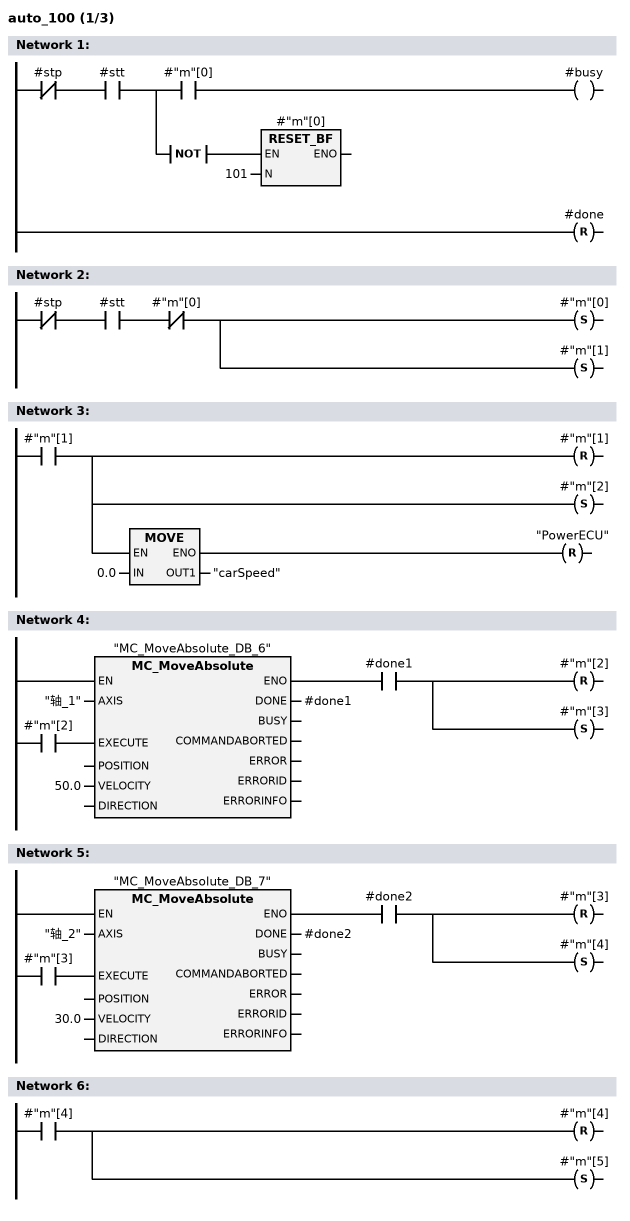
   // no SCL statement known for RBitfield: written as a call
   #_w1 := NOT #stp AND #stt;
   #busy := #_w1 AND #"m"[0];
   IF NOT #_w1 THEN RESET_BF(operand := #"m"[0], n := 101); END_IF;
   #done := FALSE;
END_REGION

REGION Network 2
   RUNG wire#powerrail
      I_Contact( #stp )
      Contact( #stt )
      I_Contact( #"m"[0] )
      wire#w1
      S_Coil( #"m"[0] )
   END_RUNG
   RUNG wire#w1
      S_Coil( #"m"[1] )
   END_RUNG
   // the same network as SCL:
   #_w1 := NOT #stp AND #stt AND NOT #"m"[0];
   IF #_w1 THEN
       #"m"[0] := TRUE;
       #"m"[1] := TRUE;
   END_IF;
END_REGION

REGION Network 3
   RUNG wire#powerrail
      Contact( #"m"[1] )
      wire#w1
      R_Coil( #"m"[1] )
   END_RUNG
   RUNG wire#w1
      S_Coil( #"m"[2] )
   END_RUNG
   RUNG wire#w1
      Move(in := 0.0, out1 => "carSpeed")
      R_Coil( "PowerECU" )
   END_RUNG
   // the same network as SCL:
   #_w1 := #"m"[1];
   IF #_w1 THEN
       #"m"[1] := FALSE;
       #"m"[2] := TRUE;
       "carSpeed" := 0.0;
       "PowerECU" := FALSE;
   END_IF;
END_REGION

REGION Network 4
   // ENO of a box is taken as its EN; it also drops when the box reports an error
   "MC_MoveAbsolute_DB_6"(Axis := "轴_1", Execute := #"m"[2], Velocity := 50.0, Done => #done1);   // MC_MoveAbsolute
   IF #done1 THEN
       #"m"[2] := FALSE;
       #"m"[3] := TRUE;
   END_IF;
END_REGION

REGION Network 5
   // ENO of a box is taken as its EN; it also drops when the box reports an error
   "MC_MoveAbsolute_DB_7"(Axis := "轴_2", Execute := #"m"[3], Velocity := 30.0, Done => #done2);   // MC_MoveAbsolute
   IF #done2 THEN
       #"m"[3] := FALSE;
       #"m"[4] := TRUE;
   END_IF;
END_REGION

REGION Network 6
   RUNG wire#powerrail
      Contact( #"m"[4] )
      wire#w1
      R_Coil( #"m"[4] )
   END_RUNG
   RUNG wire#w1
      S_Coil( #"m"[5] )
   END_RUNG
   // the same network as SCL:
   #_w1 := #"m"[4];
   IF #_w1 THEN
       #"m"[4] := FALSE;
       #"m"[5] := TRUE;
   END_IF;
END_REGION

REGION Network 7
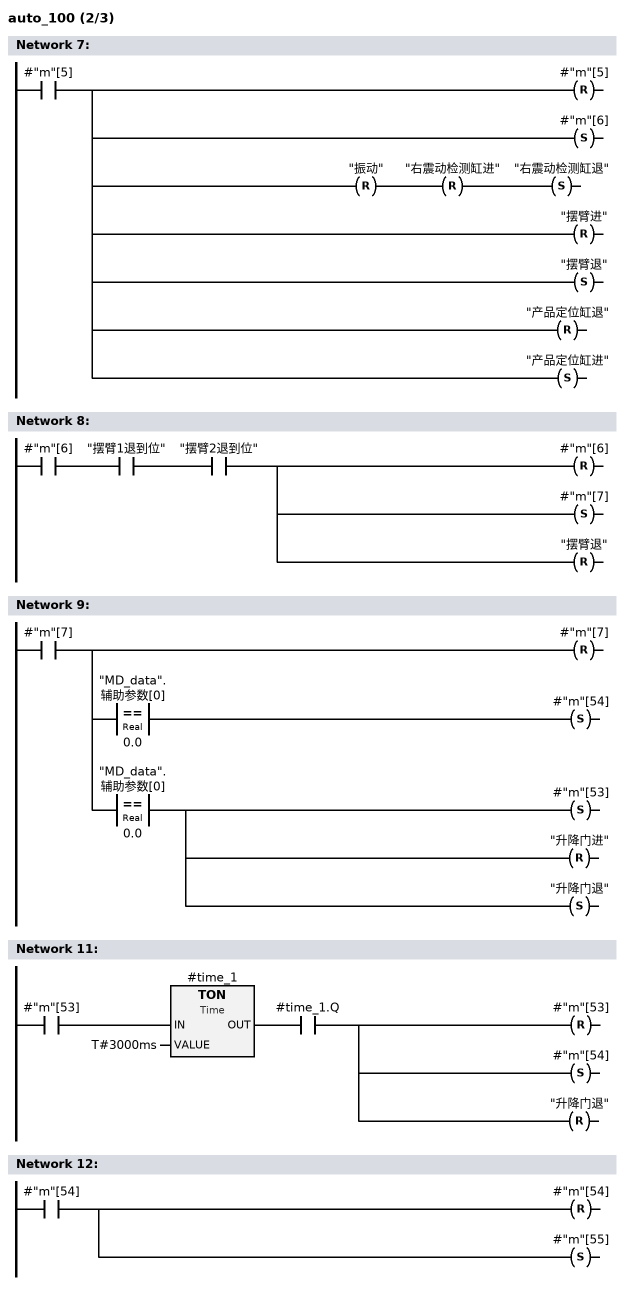
   RUNG wire#powerrail
      Contact( #"m"[5] )
      wire#w1
      R_Coil( #"m"[5] )
   END_RUNG
   RUNG wire#w1
      S_Coil( #"m"[6] )
   END_RUNG
   RUNG wire#w1
      R_Coil( "振动" )
      R_Coil( "右震动检测缸进" )
      S_Coil( "右震动检测缸退" )
   END_RUNG
   RUNG wire#w1
      R_Coil( "摆臂进" )
   END_RUNG
   RUNG wire#w1
      S_Coil( "摆臂退" )
   END_RUNG
   RUNG wire#w1
      R_Coil( "产品定位缸退" )
   END_RUNG
   RUNG wire#w1
      S_Coil( "产品定位缸进" )
   END_RUNG
   // the same network as SCL:
   #_w1 := #"m"[5];
   IF #_w1 THEN
       #"m"[5] := FALSE;
       #"m"[6] := TRUE;
       "振动" := FALSE;
       "右震动检测缸进" := FALSE;
       "右震动检测缸退" := TRUE;
       "摆臂进" := FALSE;
       "摆臂退" := TRUE;
       "产品定位缸退" := FALSE;
       "产品定位缸进" := TRUE;
   END_IF;
END_REGION

REGION Network 8
   RUNG wire#powerrail
      Contact( #"m"[6] )
      Contact( "摆臂1退到位" )
      Contact( "摆臂2退到位" )
      wire#w1
      R_Coil( #"m"[6] )
   END_RUNG
   RUNG wire#w1
      S_Coil( #"m"[7] )
   END_RUNG
   RUNG wire#w1
      R_Coil( "摆臂退" )
   END_RUNG
   // the same network as SCL:
   #_w1 := #"m"[6] AND "摆臂1退到位" AND "摆臂2退到位";
   IF #_w1 THEN
       #"m"[6] := FALSE;
       #"m"[7] := TRUE;
       "摆臂退" := FALSE;
   END_IF;
END_REGION

REGION Network 9
   RUNG wire#powerrail
      Contact( #"m"[7] )
      wire#w1
      R_Coil( #"m"[7] )
   END_RUNG
   RUNG wire#w1
      { S7_Templates := "SrcType := Real" } EQ_Contact(in1 := "MD_data".辅助参数[0], in2 := 0.0)
      S_Coil( #"m"[54] )
   END_RUNG
   RUNG wire#w1
      { S7_Templates := "SrcType := Real" } EQ_Contact(in1 := "MD_data".辅助参数[0], in2 := 0.0)
      wire#w2
      S_Coil( #"m"[53] )
   END_RUNG
   RUNG wire#w2
      R_Coil( "升降门进" )
   END_RUNG
   RUNG wire#w2
      S_Coil( "升降门退" )
   END_RUNG
   // the same network as SCL:
   #_w1 := #"m"[7];
   IF #_w1 THEN #"m"[7] := FALSE; END_IF;
   IF #_w1 AND ("MD_data".辅助参数[0] = 0.0) THEN
       #"m"[54] := TRUE;
       #"m"[53] := TRUE;
       "升降门进" := FALSE;
       "升降门退" := TRUE;
   END_IF;
END_REGION

REGION Network 11
   #time_1.TON(IN := #"m"[53], PT := T#3000ms);   // TON coil
   #_w1 := #"m"[53] AND #time_1.Q;
   IF #_w1 THEN
       #"m"[53] := FALSE;
       #"m"[54] := TRUE;
       "升降门退" := FALSE;
   END_IF;
END_REGION

REGION Network 12
   RUNG wire#powerrail
      Contact( #"m"[54] )
      wire#w1
      R_Coil( #"m"[54] )
   END_RUNG
   RUNG wire#w1
      S_Coil( #"m"[55] )
   END_RUNG
   // the same network as SCL:
   #_w1 := #"m"[54];
   IF #_w1 THEN
       #"m"[54] := FALSE;
       #"m"[55] := TRUE;
   END_IF;
END_REGION

REGION Network 14
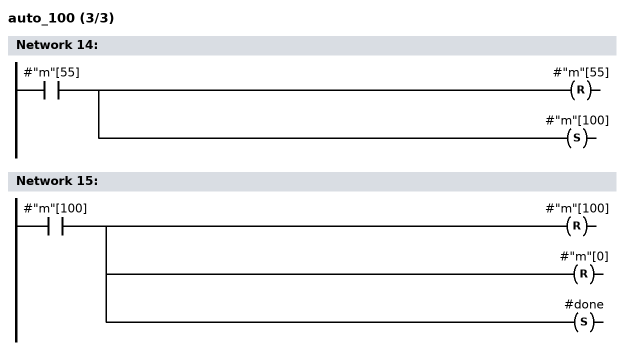
   RUNG wire#powerrail
      Contact( #"m"[55] )
      wire#w1
      R_Coil( #"m"[55] )
   END_RUNG
   RUNG wire#w1
      S_Coil( #"m"[100] )
   END_RUNG
   // the same network as SCL:
   #_w1 := #"m"[55];
   IF #_w1 THEN
       #"m"[55] := FALSE;
       #"m"[100] := TRUE;
   END_IF;
END_REGION

REGION Network 15
   RUNG wire#powerrail
      Contact( #"m"[100] )
      wire#w1
      R_Coil( #"m"[100] )
   END_RUNG
   RUNG wire#w1
      R_Coil( #"m"[0] )
   END_RUNG
   RUNG wire#w1
      S_Coil( #done )
   END_RUNG
   // the same network as SCL:
   #_w1 := #"m"[100];
   IF #_w1 THEN
       #"m"[100] := FALSE;
       #"m"[0] := FALSE;
       #done := TRUE;
   END_IF;
END_REGION
END_FUNCTION_BLOCK

FUNCTION_BLOCK "功能"   // FB14, LAD
{ S7_Optimized_Access := 'TRUE' }
VERSION : 0.1
   VAR_INPUT
      stt : Bool;
      stp : Bool;
      direction : Bool;
      speed : Real;
      angle : Real;
   END_VAR
   VAR_OUTPUT
      done : Bool;
      error : Bool;
      busy : Bool;
   END_VAR
   VAR
      "m" : Array[0..100] of Bool;
      "time" : IEC_TIMER;
      newCV : DInt;
      angleSet : Real;
      speedSet : Real;
      angleRead : Real;
      torqueOutputB : Real;
      loadOutput : Real;
      speedReal : Real;
   END_VAR
   VAR_TEMP   // added for the SCL form of the ladder/FBD networks
      _w1 : Bool;
      _w2 : Bool;
      _w3 : Bool;
      _w4 : Bool;
      _w5 : Bool;
   END_VAR
BEGIN

REGION Network 1
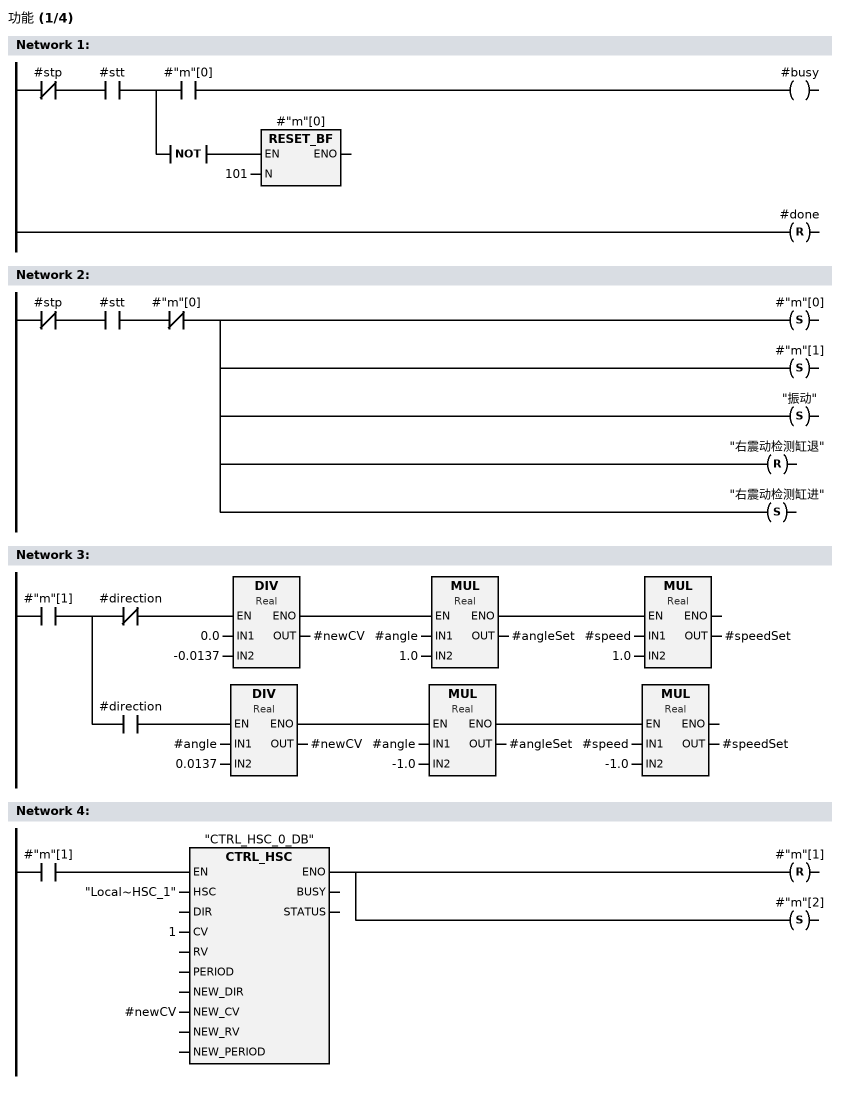
   // no SCL statement known for RBitfield: written as a call
   #_w1 := NOT #stp AND #stt;
   #busy := #_w1 AND #"m"[0];
   IF NOT #_w1 THEN RESET_BF(operand := #"m"[0], n := 101); END_IF;
   #done := FALSE;
END_REGION

REGION Network 2
   RUNG wire#powerrail
      I_Contact( #stp )
      Contact( #stt )
      I_Contact( #"m"[0] )
      wire#w1
      S_Coil( #"m"[0] )
   END_RUNG
   RUNG wire#w1
      S_Coil( #"m"[1] )
   END_RUNG
   RUNG wire#w1
      S_Coil( "振动" )
   END_RUNG
   RUNG wire#w1
      R_Coil( "右震动检测缸退" )
   END_RUNG
   RUNG wire#w1
      S_Coil( "右震动检测缸进" )
   END_RUNG
   // the same network as SCL:
   #_w1 := NOT #stp AND #stt AND NOT #"m"[0];
   IF #_w1 THEN
       #"m"[0] := TRUE;
       #"m"[1] := TRUE;
       "振动" := TRUE;
       "右震动检测缸退" := FALSE;
       "右震动检测缸进" := TRUE;
   END_IF;
END_REGION

REGION Network 3
   RUNG wire#powerrail
      Contact( #"m"[1] )
      wire#w1
      I_Contact( #direction )
      { S7_Templates := "SrcType := Real" } Div(in1 := 0.0, in2 := -0.0137, out => #newCV)
      { S7_Templates := "SrcType := Real" } Mul(in1 := #angle, in2 := 1.0, out => #angleSet)
      { S7_Templates := "SrcType := Real" } Mul(in1 := #speed, in2 := 1.0, out => #speedSet)
   END_RUNG
   RUNG wire#w1
      Contact( #direction )
      { S7_Templates := "SrcType := Real" } Div(in1 := #angle, in2 := 0.0137, out => #newCV)
      { S7_Templates := "SrcType := Real" } Mul(in1 := #angle, in2 := -1.0, out => #angleSet)
      { S7_Templates := "SrcType := Real" } Mul(in1 := #speed, in2 := -1.0, out => #speedSet)
   END_RUNG
   // the same network as SCL:
   IF #"m"[1] AND NOT #direction THEN
       #newCV := 0.0 / (-0.0137);
       #angleSet := #angle * 1.0;
       #speedSet := #speed * 1.0;
   END_IF;
   IF #"m"[1] AND #direction THEN
       #newCV := #angle / 0.0137;
       #angleSet := #angle * (-1.0);
       #speedSet := #speed * (-1.0);
   END_IF;
END_REGION

REGION Network 4
   // ENO of a box is taken as its EN; it also drops when the box reports an error
   IF #"m"[1] THEN
       "CTRL_HSC_0_DB"(HSC := "Local~HSC_1", CV := 1, NEW_CV := #newCV);   // CTRL_HSC
   END_IF;
   #_w1 := #"m"[1];
   IF #_w1 THEN
       #"m"[1] := FALSE;
       #"m"[2] := TRUE;
   END_IF;
END_REGION

REGION Network 5
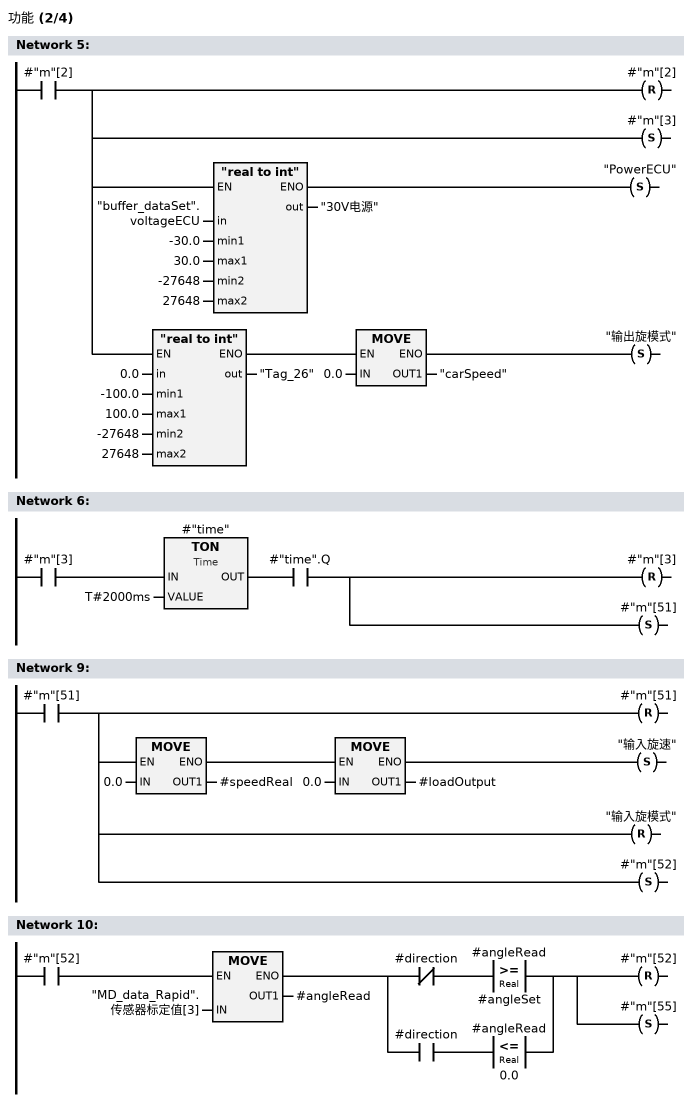
   RUNG wire#powerrail
      Contact( #"m"[2] )
      wire#w1
      R_Coil( #"m"[2] )
   END_RUNG
   RUNG wire#w1
      S_Coil( #"m"[3] )
   END_RUNG
   RUNG wire#w1
      "real to int"(in := "buffer_dataSet".voltageECU, min1 := -30.0, max1 := 30.0, min2 := -27648, max2 := 27648, out => "30V电源")
      S_Coil( "PowerECU" )
   END_RUNG
   RUNG wire#w1
      "real to int"(in := 0.0, min1 := -100.0, max1 := 100.0, min2 := -27648, max2 := 27648, out => "Tag_26")
      Move(in := 0.0, out1 => "carSpeed")
      S_Coil( "输出旋模式" )
   END_RUNG
   // the same network as SCL:
   #_w1 := #"m"[2];
   IF #_w1 THEN
       #"m"[2] := FALSE;
       #"m"[3] := TRUE;
   END_IF;
   "real to int"(EN := #_w1,
                 in := "buffer_dataSet".voltageECU,
                 min1 := -30.0,
                 max1 := 30.0,
                 min2 := -27648,
                 max2 := 27648,
                 out => "30V电源",
                 ENO => #_w2);
   IF #_w2 THEN "PowerECU" := TRUE; END_IF;
   "real to int"(EN := #_w1,
                 in := 0.0,
                 min1 := -100.0,
                 max1 := 100.0,
                 min2 := -27648,
                 max2 := 27648,
                 out => "Tag_26",
                 ENO => #_w3);
   IF #_w3 THEN
       "carSpeed" := 0.0;
       "输出旋模式" := TRUE;
   END_IF;
END_REGION

REGION Network 6
   #"time".TON(IN := #"m"[3], PT := T#2000ms);   // TON coil
   #_w1 := #"m"[3] AND #"time".Q;
   IF #_w1 THEN
       #"m"[3] := FALSE;
       #"m"[51] := TRUE;
   END_IF;
END_REGION

REGION Network 9
   RUNG wire#powerrail
      Contact( #"m"[51] )
      wire#w1
      R_Coil( #"m"[51] )
   END_RUNG
   RUNG wire#w1
      Move(in := 0.0, out1 => #speedReal)
      Move(in := 0.0, out1 => #loadOutput)
      S_Coil( "输入旋速" )
   END_RUNG
   RUNG wire#w1
      R_Coil( "输入旋模式" )
   END_RUNG
   RUNG wire#w1
      S_Coil( #"m"[52] )
   END_RUNG
   // the same network as SCL:
   #_w1 := #"m"[51];
   IF #_w1 THEN
       #"m"[51] := FALSE;
       #speedReal := 0.0;
       #loadOutput := 0.0;
       "输入旋速" := TRUE;
       "输入旋模式" := FALSE;
       #"m"[52] := TRUE;
   END_IF;
END_REGION

REGION Network 10
   RUNG wire#powerrail
      Contact( #"m"[52] )
      Move(in := "MD_data_Rapid".传感器标定值[3], out1 => #angleRead)
      wire#w1
      I_Contact( #direction )
      { S7_Templates := "SrcType := Real" } GE_Contact(in1 := #angleRead, in2 := #angleSet)
      wire#w2
      R_Coil( #"m"[52] )
   END_RUNG
   RUNG wire#w1
      Contact( #direction )
      { S7_Templates := "SrcType := Real" } LE_Contact(in1 := #angleRead, in2 := 0.0)
   END_RUNG wire#w2
   RUNG wire#w2
      S_Coil( #"m"[55] )
   END_RUNG
   // the same network as SCL:
   IF #"m"[52] THEN #angleRead := "MD_data_Rapid".传感器标定值[3]; END_IF;
   #_w1 := #"m"[52] AND ((NOT #direction AND (#angleRead >= #angleSet)) OR (#direction AND (#angleRead <= 0.0)));
   IF #_w1 THEN
       #"m"[52] := FALSE;
       #"m"[55] := TRUE;
   END_IF;
END_REGION

REGION Network 11
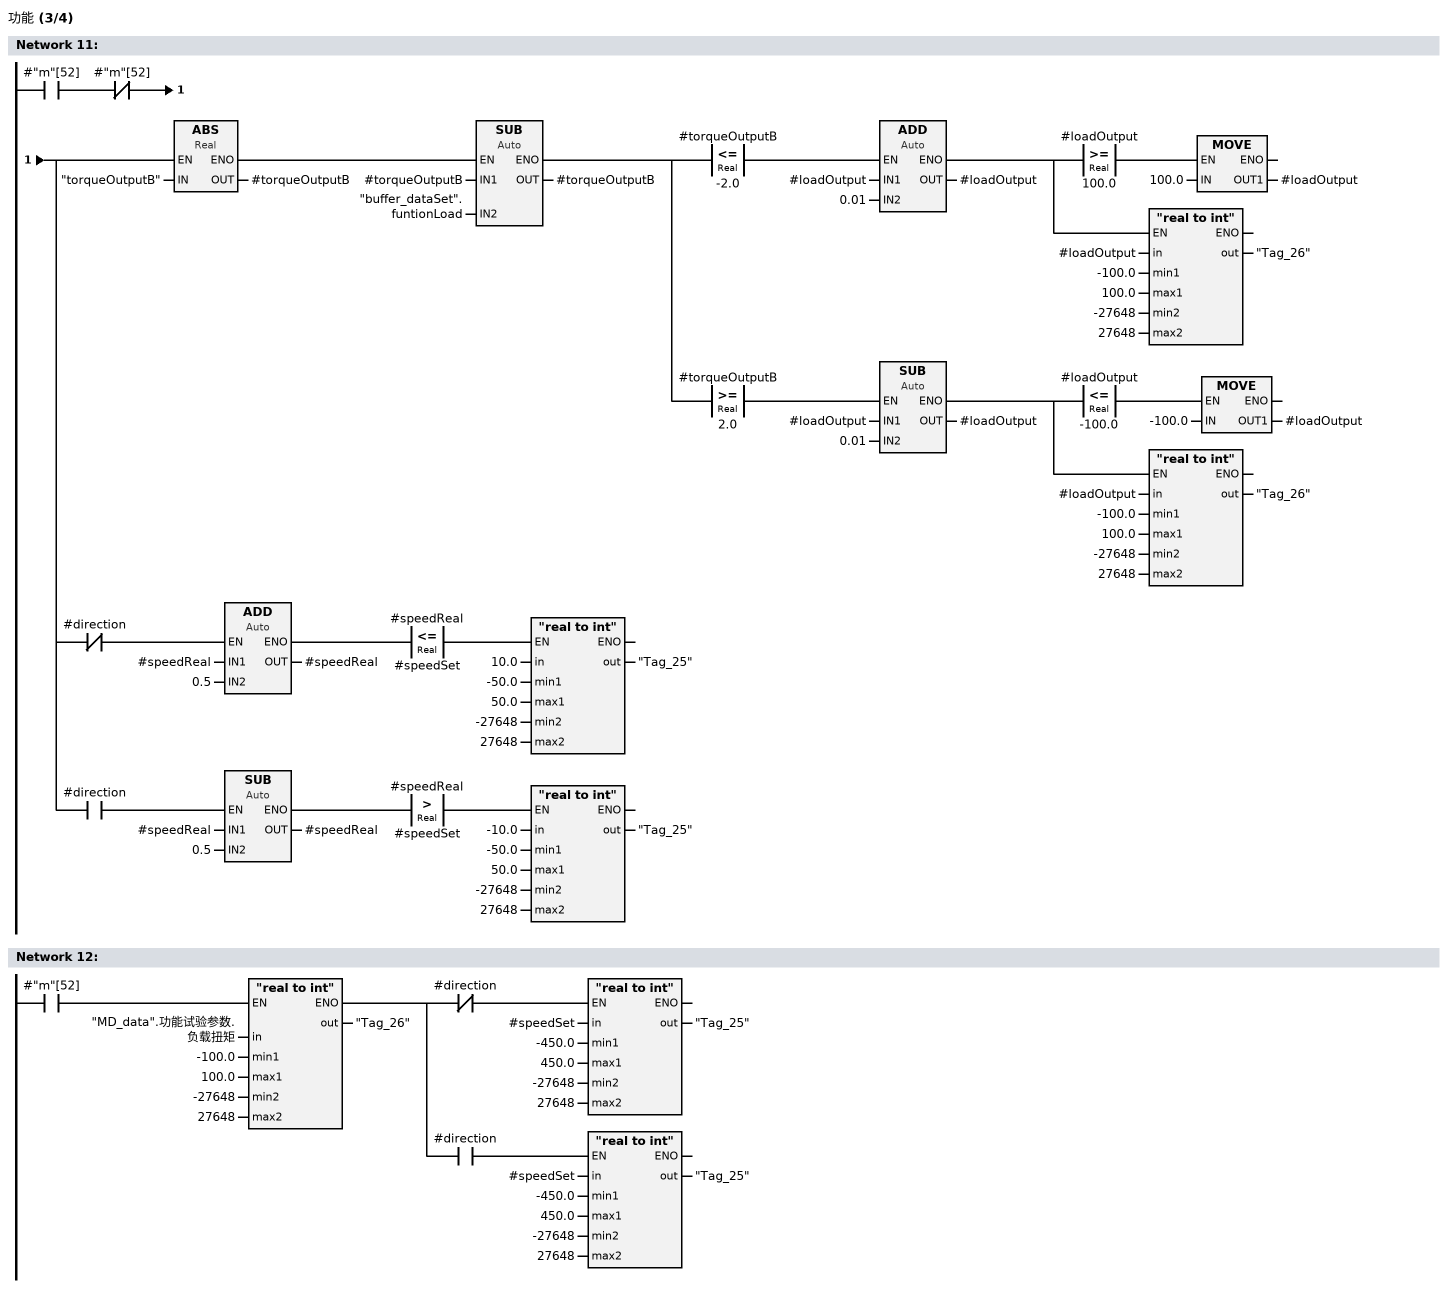
   RUNG wire#powerrail
      Contact( #"m"[52] )
      I_Contact( #"m"[52] )
      wire#w1
      { S7_Templates := "SrcType := Real" } Abs(in := "torqueOutputB", out => #torqueOutputB)
      Sub(in1 := #torqueOutputB, in2 := "buffer_dataSet".funtionLoad, out => #torqueOutputB)
      wire#w2
      { S7_Templates := "SrcType := Real" } LE_Contact(in1 := #torqueOutputB, in2 := -2.0)
      Add(in1 := #loadOutput, in2 := 0.01, out => #loadOutput)
      wire#w3
      { S7_Templates := "SrcType := Real" } GE_Contact(in1 := #loadOutput, in2 := 100.0)
      Move(in := 100.0, out1 => #loadOutput)
   END_RUNG
   RUNG wire#w3
      "real to int"(in := #loadOutput, min1 := -100.0, max1 := 100.0, min2 := -27648, max2 := 27648, out => "Tag_26")
   END_RUNG
   RUNG wire#w2
      { S7_Templates := "SrcType := Real" } GE_Contact(in1 := #torqueOutputB, in2 := 2.0)
      Sub(in1 := #loadOutput, in2 := 0.01, out => #loadOutput)
      wire#w4
      { S7_Templates := "SrcType := Real" } LE_Contact(in1 := #loadOutput, in2 := -100.0)
      Move(in := -100.0, out1 => #loadOutput)
   END_RUNG
   RUNG wire#w4
      "real to int"(in := #loadOutput, min1 := -100.0, max1 := 100.0, min2 := -27648, max2 := 27648, out => "Tag_26")
   END_RUNG
   RUNG wire#w1
      I_Contact( #direction )
      Add(in1 := #speedReal, in2 := 0.5, out => #speedReal)
      { S7_Templates := "SrcType := Real" } LE_Contact(in1 := #speedReal, in2 := #speedSet)
      "real to int"(in := 10.0, min1 := -50.0, max1 := 50.0, min2 := -27648, max2 := 27648, out => "Tag_25")
   END_RUNG
   RUNG wire#w1
      Contact( #direction )
      Sub(in1 := #speedReal, in2 := 0.5, out => #speedReal)
      { S7_Templates := "SrcType := Real" } GT_Contact(in1 := #speedReal, in2 := #speedSet)
      "real to int"(in := -10.0, min1 := -50.0, max1 := 50.0, min2 := -27648, max2 := 27648, out => "Tag_25")
   END_RUNG
   // the same network as SCL:
   #_w1 := #"m"[52] AND NOT #"m"[52];
   IF #_w1 THEN
       #torqueOutputB := ABS("torqueOutputB");
       #torqueOutputB := #torqueOutputB - "buffer_dataSet".funtionLoad;
   END_IF;
   #_w2 := #_w1 AND (#torqueOutputB <= (-2.0));
   IF #_w2 THEN #loadOutput := #loadOutput + 0.01; END_IF;
   IF #_w2 AND (#loadOutput >= 100.0) THEN #loadOutput := 100.0; END_IF;
   IF #_w2 THEN
       "real to int"(in := #loadOutput,
                     min1 := -100.0,
                     max1 := 100.0,
                     min2 := -27648,
                     max2 := 27648,
                     out => "Tag_26");
   END_IF;
   #_w3 := #_w1 AND (#torqueOutputB >= 2.0);
   IF #_w3 THEN #loadOutput := #loadOutput - 0.01; END_IF;
   IF #_w3 AND (#loadOutput <= (-100.0)) THEN #loadOutput := -100.0; END_IF;
   IF #_w3 THEN
       "real to int"(in := #loadOutput,
                     min1 := -100.0,
                     max1 := 100.0,
                     min2 := -27648,
                     max2 := 27648,
                     out => "Tag_26");
   END_IF;
   #_w4 := #_w1 AND NOT #direction;
   IF #_w4 THEN #speedReal := #speedReal + 0.5; END_IF;
   IF #_w4 AND (#speedReal <= #speedSet) THEN
       "real to int"(in := 10.0, min1 := -50.0, max1 := 50.0, min2 := -27648, max2 := 27648, out => "Tag_25");
   END_IF;
   #_w5 := #_w1 AND #direction;
   IF #_w5 THEN #speedReal := #speedReal - 0.5; END_IF;
   IF #_w5 AND (#speedReal > #speedSet) THEN
       "real to int"(in := -10.0, min1 := -50.0, max1 := 50.0, min2 := -27648, max2 := 27648, out => "Tag_25");
   END_IF;
END_REGION

REGION Network 12
   RUNG wire#powerrail
      Contact( #"m"[52] )
      "real to int"(in := "MD_data".功能试验参数.负载扭矩, min1 := -100.0, max1 := 100.0, min2 := -27648, max2 := 27648, out => "Tag_26")
      wire#w1
      I_Contact( #direction )
      "real to int"(in := #speedSet, min1 := -450.0, max1 := 450.0, min2 := -27648, max2 := 27648, out => "Tag_25")
   END_RUNG
   RUNG wire#w1
      Contact( #direction )
      "real to int"(in := #speedSet, min1 := -450.0, max1 := 450.0, min2 := -27648, max2 := 27648, out => "Tag_25")
   END_RUNG
   // the same network as SCL:
   "real to int"(EN := #"m"[52],
                 in := "MD_data".功能试验参数.负载扭矩,
                 min1 := -100.0,
                 max1 := 100.0,
                 min2 := -27648,
                 max2 := 27648,
                 out => "Tag_26",
                 ENO => #_w1);
   IF #_w1 AND NOT #direction THEN
       "real to int"(in := #speedSet, min1 := -450.0, max1 := 450.0, min2 := -27648, max2 := 27648, out => "Tag_25");
   END_IF;
   IF #_w1 AND #direction THEN
       "real to int"(in := #speedSet, min1 := -450.0, max1 := 450.0, min2 := -27648, max2 := 27648, out => "Tag_25");
   END_IF;
END_REGION

REGION Network 13
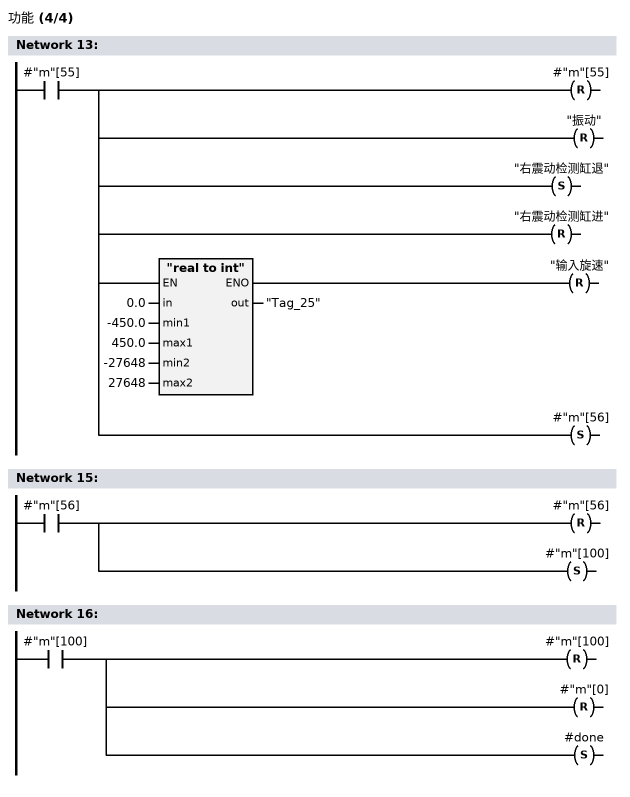
   RUNG wire#powerrail
      Contact( #"m"[55] )
      wire#w1
      R_Coil( #"m"[55] )
   END_RUNG
   RUNG wire#w1
      R_Coil( "振动" )
   END_RUNG
   RUNG wire#w1
      S_Coil( "右震动检测缸退" )
   END_RUNG
   RUNG wire#w1
      R_Coil( "右震动检测缸进" )
   END_RUNG
   RUNG wire#w1
      "real to int"(in := 0.0, min1 := -450.0, max1 := 450.0, min2 := -27648, max2 := 27648, out => "Tag_25")
      R_Coil( "输入旋速" )
   END_RUNG
   RUNG wire#w1
      S_Coil( #"m"[56] )
   END_RUNG
   // the same network as SCL:
   #_w1 := #"m"[55];
   IF #_w1 THEN
       #"m"[55] := FALSE;
       "振动" := FALSE;
       "右震动检测缸退" := TRUE;
       "右震动检测缸进" := FALSE;
   END_IF;
   "real to int"(EN := #_w1,
                 in := 0.0,
                 min1 := -450.0,
                 max1 := 450.0,
                 min2 := -27648,
                 max2 := 27648,
                 out => "Tag_25",
                 ENO => #_w2);
   IF #_w2 THEN "输入旋速" := FALSE; END_IF;
   IF #_w1 THEN #"m"[56] := TRUE; END_IF;
END_REGION

REGION Network 15
   RUNG wire#powerrail
      Contact( #"m"[56] )
      wire#w1
      R_Coil( #"m"[56] )
   END_RUNG
   RUNG wire#w1
      S_Coil( #"m"[100] )
   END_RUNG
   // the same network as SCL:
   #_w1 := #"m"[56];
   IF #_w1 THEN
       #"m"[56] := FALSE;
       #"m"[100] := TRUE;
   END_IF;
END_REGION

REGION Network 16
   RUNG wire#powerrail
      Contact( #"m"[100] )
      wire#w1
      R_Coil( #"m"[100] )
   END_RUNG
   RUNG wire#w1
      R_Coil( #"m"[0] )
   END_RUNG
   RUNG wire#w1
      S_Coil( #done )
   END_RUNG
   // the same network as SCL:
   #_w1 := #"m"[100];
   IF #_w1 THEN
       #"m"[100] := FALSE;
       #"m"[0] := FALSE;
       #done := TRUE;
   END_IF;
END_REGION
END_FUNCTION_BLOCK

FUNCTION_BLOCK "找零"   // FB15, LAD
{ S7_Optimized_Access := 'TRUE' }
VERSION : 0.1
   VAR_INPUT
      stp : Bool;
      stt : Bool;
      direction : Bool;
      speed : Real;
      torque : Real;
   END_VAR
   VAR_OUTPUT
      done : Bool;
      error : Bool;
      busy : Bool;
   END_VAR
   VAR
      "m" : Array[0..10] of Bool;
      speedSet : Real;
      torqueSet : Real;
      IEC_Timer_0_Instance : TON_TIME;
   END_VAR
   VAR_TEMP   // added for the SCL form of the ladder/FBD networks
      _w1 : Bool;
      _w2 : Bool;
   END_VAR
BEGIN

REGION Network 1
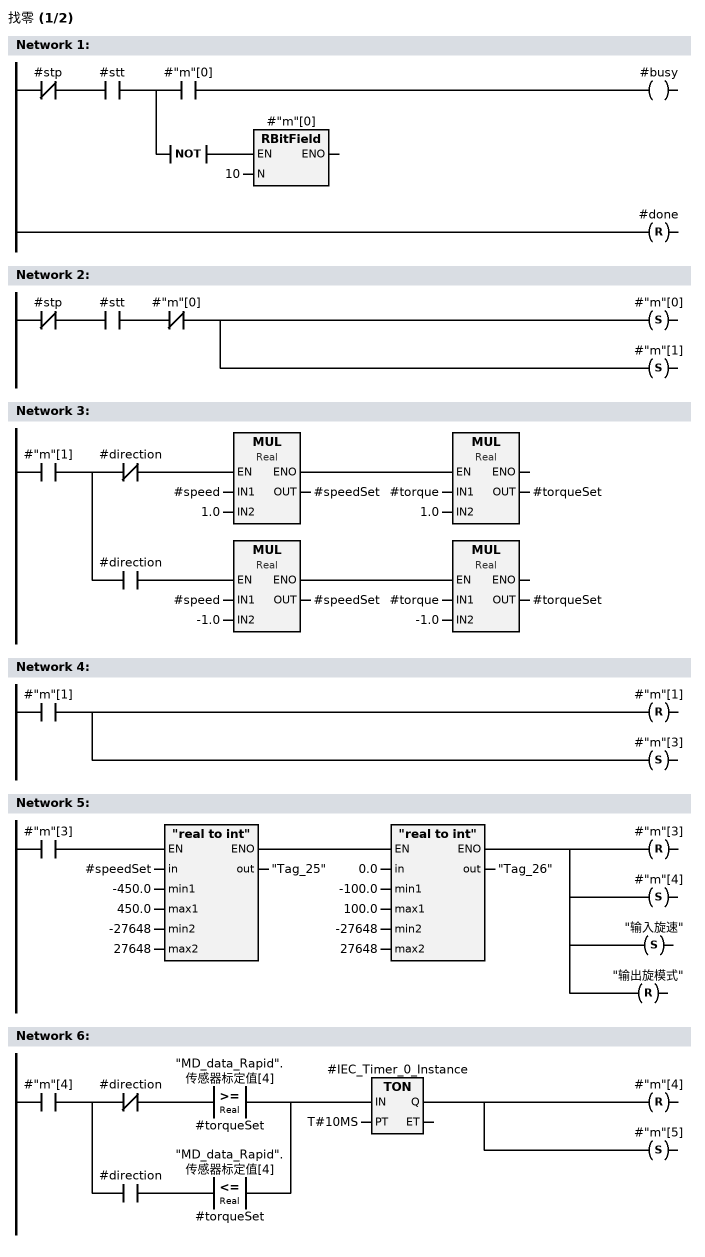
   // no SCL statement known for RBitField: written as a call
   #_w1 := NOT #stp AND #stt;
   #busy := #_w1 AND #"m"[0];
   IF NOT #_w1 THEN RBitField(n := 10, operand := #"m"[0]); END_IF;
   #done := FALSE;
END_REGION

REGION Network 2
   RUNG wire#powerrail
      I_Contact( #stp )
      Contact( #stt )
      I_Contact( #"m"[0] )
      wire#w1
      S_Coil( #"m"[0] )
   END_RUNG
   RUNG wire#w1
      S_Coil( #"m"[1] )
   END_RUNG
   // the same network as SCL:
   #_w1 := NOT #stp AND #stt AND NOT #"m"[0];
   IF #_w1 THEN
       #"m"[0] := TRUE;
       #"m"[1] := TRUE;
   END_IF;
END_REGION

REGION Network 3
   RUNG wire#powerrail
      Contact( #"m"[1] )
      wire#w1
      I_Contact( #direction )
      { S7_Templates := "SrcType := Real" } Mul(in1 := #speed, in2 := 1.0, out => #speedSet)
      { S7_Templates := "SrcType := Real" } Mul(in1 := #torque, in2 := 1.0, out => #torqueSet)
   END_RUNG
   RUNG wire#w1
      Contact( #direction )
      { S7_Templates := "SrcType := Real" } Mul(in1 := #speed, in2 := -1.0, out => #speedSet)
      { S7_Templates := "SrcType := Real" } Mul(in1 := #torque, in2 := -1.0, out => #torqueSet)
   END_RUNG
   // the same network as SCL:
   IF #"m"[1] AND NOT #direction THEN
       #speedSet := #speed * 1.0;
       #torqueSet := #torque * 1.0;
   END_IF;
   IF #"m"[1] AND #direction THEN
       #speedSet := #speed * (-1.0);
       #torqueSet := #torque * (-1.0);
   END_IF;
END_REGION

REGION Network 4
   RUNG wire#powerrail
      Contact( #"m"[1] )
      wire#w1
      R_Coil( #"m"[1] )
   END_RUNG
   RUNG wire#w1
      S_Coil( #"m"[3] )
   END_RUNG
   // the same network as SCL:
   #_w1 := #"m"[1];
   IF #_w1 THEN
       #"m"[1] := FALSE;
       #"m"[3] := TRUE;
   END_IF;
END_REGION

REGION Network 5
   RUNG wire#powerrail
      Contact( #"m"[3] )
      "real to int"(in := #speedSet, min1 := -450.0, max1 := 450.0, min2 := -27648, max2 := 27648, out => "Tag_25")
      "real to int"(in := 0.0, min1 := -100.0, max1 := 100.0, min2 := -27648, max2 := 27648, out => "Tag_26")
      wire#w1
      R_Coil( #"m"[3] )
   END_RUNG
   RUNG wire#w1
      S_Coil( #"m"[4] )
   END_RUNG
   RUNG wire#w1
      S_Coil( "输入旋速" )
   END_RUNG
   RUNG wire#w1
      R_Coil( "输出旋模式" )
   END_RUNG
   // the same network as SCL:
   "real to int"(EN := #"m"[3],
                 in := #speedSet,
                 min1 := -450.0,
                 max1 := 450.0,
                 min2 := -27648,
                 max2 := 27648,
                 out => "Tag_25",
                 ENO => #_w1);
   "real to int"(EN := #_w1,
                 in := 0.0,
                 min1 := -100.0,
                 max1 := 100.0,
                 min2 := -27648,
                 max2 := 27648,
                 out => "Tag_26",
                 ENO => #_w2);
   IF #_w2 THEN
       #"m"[3] := FALSE;
       #"m"[4] := TRUE;
       "输入旋速" := TRUE;
       "输出旋模式" := FALSE;
   END_IF;
END_REGION

REGION Network 6
   #IEC_Timer_0_Instance(IN := #"m"[4] AND ((NOT #direction AND ("MD_data_Rapid".传感器标定值[4] >= #torqueSet)) OR (#direction AND ("MD_data_Rapid".传感器标定值[4] <= #torqueSet))),   // TON
                         PT := T#10MS);
   IF #IEC_Timer_0_Instance.Q THEN
       #"m"[4] := FALSE;
       #"m"[5] := TRUE;
   END_IF;
END_REGION

REGION Network 7
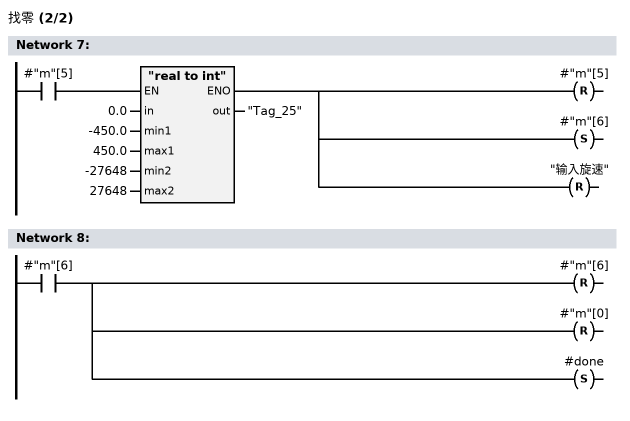
   RUNG wire#powerrail
      Contact( #"m"[5] )
      "real to int"(in := 0.0, min1 := -450.0, max1 := 450.0, min2 := -27648, max2 := 27648, out => "Tag_25")
      wire#w1
      R_Coil( #"m"[5] )
   END_RUNG
   RUNG wire#w1
      S_Coil( #"m"[6] )
   END_RUNG
   RUNG wire#w1
      R_Coil( "输入旋速" )
   END_RUNG
   // the same network as SCL:
   "real to int"(EN := #"m"[5],
                 in := 0.0,
                 min1 := -450.0,
                 max1 := 450.0,
                 min2 := -27648,
                 max2 := 27648,
                 out => "Tag_25",
                 ENO => #_w1);
   IF #_w1 THEN
       #"m"[5] := FALSE;
       #"m"[6] := TRUE;
       "输入旋速" := FALSE;
   END_IF;
END_REGION

REGION Network 8
   RUNG wire#powerrail
      Contact( #"m"[6] )
      wire#w1
      R_Coil( #"m"[6] )
   END_RUNG
   RUNG wire#w1
      R_Coil( #"m"[0] )
   END_RUNG
   RUNG wire#w1
      S_Coil( #done )
   END_RUNG
   // the same network as SCL:
   #_w1 := #"m"[6];
   IF #_w1 THEN
       #"m"[6] := FALSE;
       #"m"[0] := FALSE;
       #done := TRUE;
   END_IF;
END_REGION
END_FUNCTION_BLOCK

FUNCTION "Axis_5_home" : Void   // FC1, LAD
{ S7_Optimized_Access := 'FALSE' }
VERSION : 0.1
   VAR_TEMP
      temp_1 : Bool;
   END_VAR
BEGIN

REGION Network 2
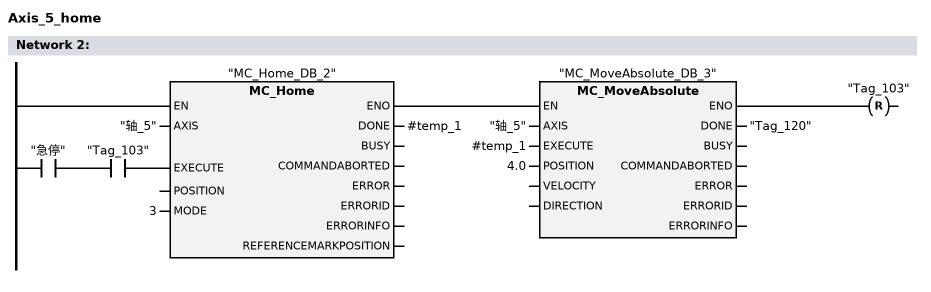
   // ENO of a box is taken as its EN; it also drops when the box reports an error
   "MC_Home_DB_2"(Axis := "轴_5", Execute := "急停" AND "Tag_103", Mode := 3, Done => #temp_1);   // MC_Home
   "MC_MoveAbsolute_DB_3"(Axis := "轴_5", Execute := #temp_1, Position := 4.0, Done => "Tag_120");   // MC_MoveAbsolute
   "Tag_103" := FALSE;
END_REGION
END_FUNCTION

FUNCTION "to angle" : Void   // FC2, LAD
{ S7_Optimized_Access := 'TRUE' }
VERSION : 0.1
   VAR_INPUT
      value : DInt;
      factor : Real;
   END_VAR
   VAR_OUTPUT
      angle : Real;
   END_VAR
BEGIN

REGION Network 1
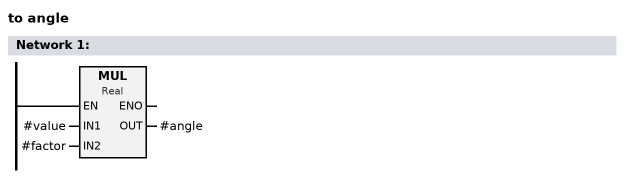
   RUNG wire#powerrail
      { S7_Templates := "SrcType := Real" } Mul(in1 := #value, in2 := #factor, out => #angle)
   END_RUNG
   // the same network as SCL:
   #angle := #value * #factor;
END_REGION
END_FUNCTION

FUNCTION "int to real" : Void   // FC3, LAD
{ S7_Optimized_Access := 'TRUE' }
VERSION : 0.1
   VAR_INPUT
      vaule : Int;
      maxOut : Real;
   END_VAR
   VAR_OUTPUT
      out : Real;
   END_VAR
   VAR_TEMP
      real_i : Real;
      real_q : Real;
      minOut : Real;
   END_VAR
BEGIN

REGION Network 1
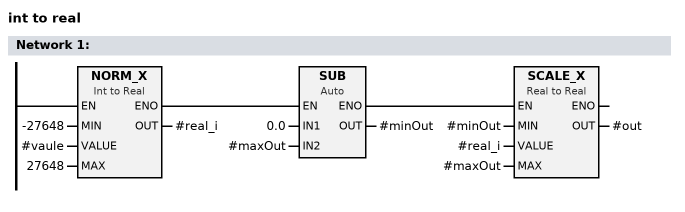
   RUNG wire#powerrail
      { S7_Templates := "[SrcType := Int, DestType := Real]" } Normalize(min := -27648, value := #vaule, max := 27648, out => #real_i)
      Sub(in1 := 0.0, in2 := #maxOut, out => #minOut)
      { S7_Templates := "[SrcType := Real, DestType := Real]" } Scale(min := #minOut, value := #real_i, max := #maxOut, out => #out)
   END_RUNG
   // the same network as SCL:
   #real_i := NORM_X(MIN := -27648, VALUE := #vaule, MAX := 27648);
   #minOut := 0.0 - #maxOut;
   #out := SCALE_X(MIN := #minOut, VALUE := #real_i, MAX := #maxOut);
END_REGION
END_FUNCTION

FUNCTION "real to int" : Void   // FC4, LAD
{ S7_Optimized_Access := 'TRUE' }
VERSION : 0.1
   VAR_INPUT
      in : Real;
      min1 : Real;
      max1 : Real;
      min2 : Int;
      max2 : Int;
   END_VAR
   VAR_OUTPUT
      out : Int;
   END_VAR
   VAR_TEMP
      real_i : Real;
      real_q : Real;
   END_VAR
BEGIN

REGION Network 1
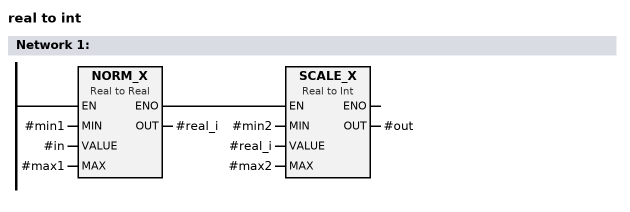
   RUNG wire#powerrail
      { S7_Templates := "[SrcType := Real, DestType := Real]" } Normalize(min := #min1, value := #in, max := #max1, out => #real_i)
      { S7_Templates := "[SrcType := Real, DestType := Int]" } Scale(min := #min2, value := #real_i, max := #max2, out => #out)
   END_RUNG
   // the same network as SCL:
   #real_i := NORM_X(MIN := #min1, VALUE := #in, MAX := #max1);
   #out := SCALE_X(MIN := #min2, VALUE := #real_i, MAX := #max2);
END_REGION
END_FUNCTION

ORGANIZATION_BLOCK "Main"   // OB1, LAD, ProgramCycle
TITLE = "Main Program Sweep (Cycle)"
{ S7_Optimized_Access := 'TRUE' }
VERSION : 0.1
   VAR_INPUT
      Initial_Call : Bool;   // Initial call of this OB
      Remanence : Bool;   // =True, if remanent data are available
   END_VAR
   VAR_TEMP
      X : UInt;
      Y : Real;
      busy : Bool;
      done : Bool;
      speed : Real;
      angle_m : Real;
      value : Real;
      value_1 : Real;
      value_2 : Real;
      value_3 : Real;
      temp_t1 : Real;
      temp_t2 : Real;
      temp_t3 : Real;
      sign : Word;
      ret_val : Int;
   END_VAR
   VAR_TEMP   // added for the SCL form of the ladder/FBD networks
      _w1 : Bool;
      _w2 : Bool;
      _w3 : Bool;
      _w4 : Bool;
      _w5 : Bool;
      _w6 : Bool;
   END_VAR
BEGIN

REGION Network 1
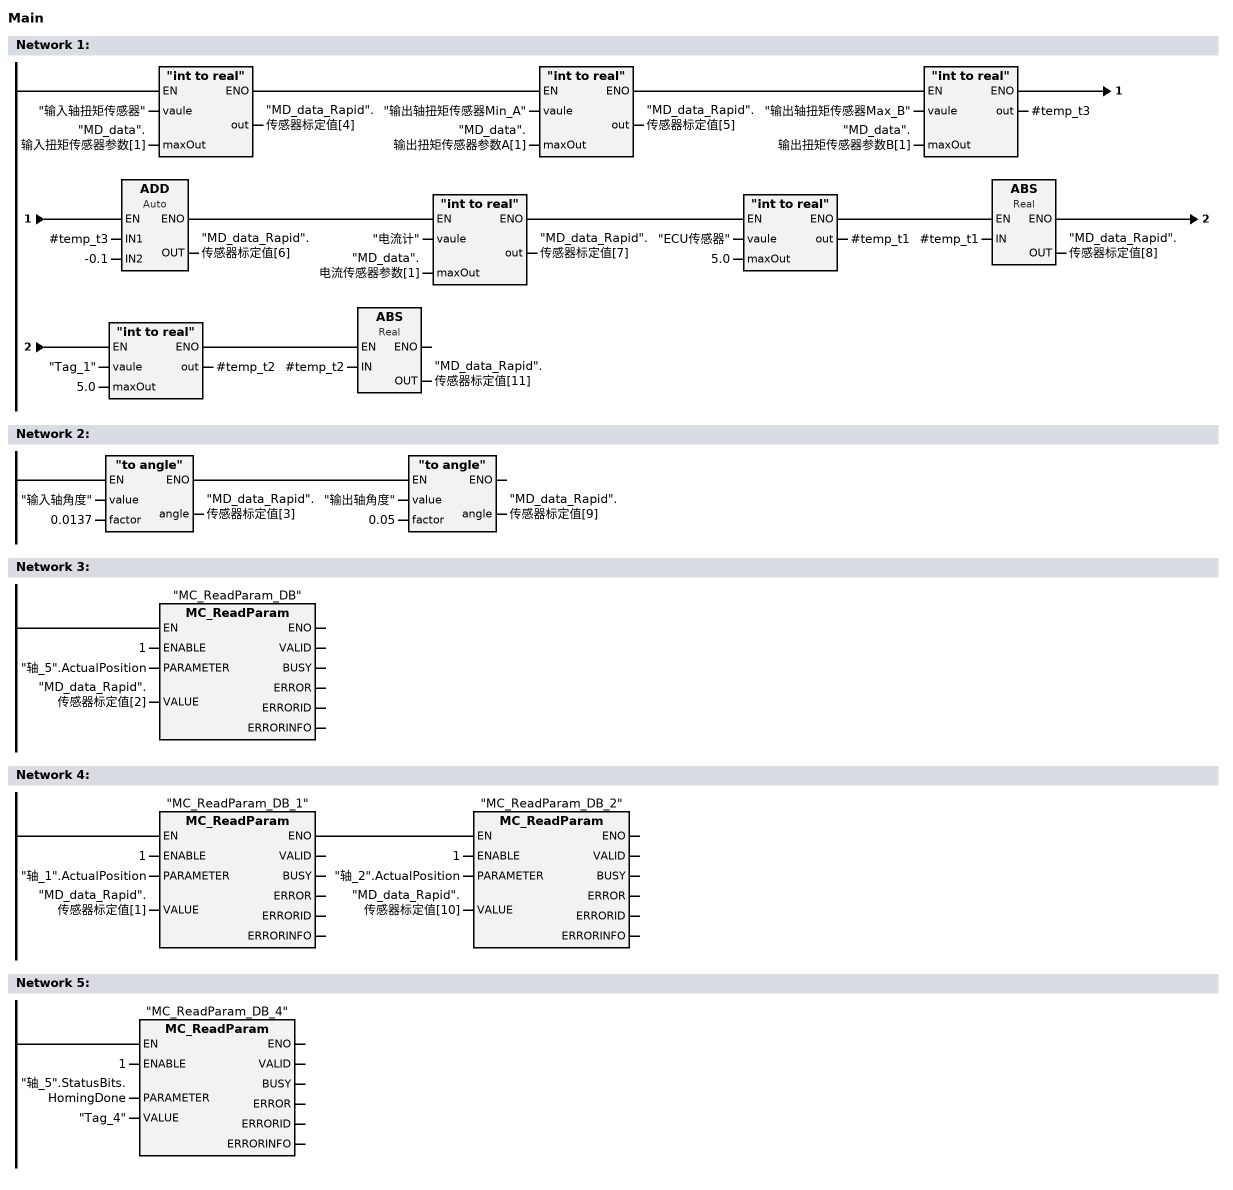
   RUNG wire#powerrail
      "int to real"(vaule := "输入轴扭矩传感器", maxOut := "MD_data".输入扭矩传感器参数[1], out => "MD_data_Rapid".传感器标定值[4])
      "int to real"(vaule := "输出轴扭矩传感器Min_A", maxOut := "MD_data".输出扭矩传感器参数A[1], out => "MD_data_Rapid".传感器标定值[5])
      "int to real"(vaule := "输出轴扭矩传感器Max_B", maxOut := "MD_data".输出扭矩传感器参数B[1], out => #temp_t3)
      Add(in1 := #temp_t3, in2 := -0.1, out => "MD_data_Rapid".传感器标定值[6])
      "int to real"(vaule := "电流计", maxOut := "MD_data".电流传感器参数[1], out => "MD_data_Rapid".传感器标定值[7])
      "int to real"(vaule := "ECU传感器", maxOut := 5.0, out => #temp_t1)
      { S7_Templates := "SrcType := Real" } Abs(in := #temp_t1, out => "MD_data_Rapid".传感器标定值[8])
      "int to real"(vaule := "Tag_1", maxOut := 5.0, out => #temp_t2)
      { S7_Templates := "SrcType := Real" } Abs(in := #temp_t2, out => "MD_data_Rapid".传感器标定值[11])
   END_RUNG
   // the same network as SCL:
   "int to real"(vaule := "输入轴扭矩传感器",
                 maxOut := "MD_data".输入扭矩传感器参数[1],
                 out => "MD_data_Rapid".传感器标定值[4],
                 ENO => #_w1);
   "int to real"(EN := #_w1,
                 vaule := "输出轴扭矩传感器Min_A",
                 maxOut := "MD_data".输出扭矩传感器参数A[1],
                 out => "MD_data_Rapid".传感器标定值[5],
                 ENO => #_w2);
   "int to real"(EN := #_w2,
                 vaule := "输出轴扭矩传感器Max_B",
                 maxOut := "MD_data".输出扭矩传感器参数B[1],
                 out => #temp_t3,
                 ENO => #_w3);
   IF #_w3 THEN "MD_data_Rapid".传感器标定值[6] := #temp_t3 + (-0.1); END_IF;
   "int to real"(EN := #_w3,
                 vaule := "电流计",
                 maxOut := "MD_data".电流传感器参数[1],
                 out => "MD_data_Rapid".传感器标定值[7],
                 ENO => #_w4);
   "int to real"(EN := #_w4, vaule := "ECU传感器", maxOut := 5.0, out => #temp_t1, ENO => #_w5);
   IF #_w5 THEN "MD_data_Rapid".传感器标定值[8] := ABS(#temp_t1); END_IF;
   "int to real"(EN := #_w5, vaule := "Tag_1", maxOut := 5.0, out => #temp_t2, ENO => #_w6);
   IF #_w6 THEN "MD_data_Rapid".传感器标定值[11] := ABS(#temp_t2); END_IF;
END_REGION

REGION Network 2
   RUNG wire#powerrail
      "to angle"(value := "输入轴角度", factor := 0.0137, angle => "MD_data_Rapid".传感器标定值[3])
      "to angle"(value := "输出轴角度", factor := 0.05, angle => "MD_data_Rapid".传感器标定值[9])
   END_RUNG
   // the same network as SCL:
   "to angle"(value := "输入轴角度", factor := 0.0137, angle => "MD_data_Rapid".传感器标定值[3], ENO => #_w1);
   IF #_w1 THEN "to angle"(value := "输出轴角度", factor := 0.05, angle => "MD_data_Rapid".传感器标定值[9]); END_IF;
END_REGION

REGION Network 3
   "MC_ReadParam_DB"(Enable := 1, Parameter := "轴_5".ActualPosition, Value := "MD_data_Rapid".传感器标定值[2]);   // MC_ReadParam
END_REGION

REGION Network 4
   // ENO of a box is taken as its EN; it also drops when the box reports an error
   "MC_ReadParam_DB_1"(Enable := 1, Parameter := "轴_1".ActualPosition, Value := "MD_data_Rapid".传感器标定值[1]);   // MC_ReadParam
   "MC_ReadParam_DB_2"(Enable := 1, Parameter := "轴_2".ActualPosition, Value := "MD_data_Rapid".传感器标定值[10]);   // MC_ReadParam
END_REGION

REGION Network 5
   "MC_ReadParam_DB_4"(Enable := 1, Parameter := "轴_5".StatusBits.HomingDone, Value := "Tag_4");   // MC_ReadParam
END_REGION
END_ORGANIZATION_BLOCK

ORGANIZATION_BLOCK "Cyclic interrupt_10ms"   // OB30, LAD, CyclicInterrupt
{ S7_Optimized_Access := 'TRUE' }
VERSION : 0.1
   VAR_INPUT
      Initial_Call : Bool;   // Initial call of this OB
      Event_Count : Int;   // Events discarded
   END_VAR
   VAR_TEMP
      done : Bool;
      done_1 : Bool;
      done_2 : Bool;
      busy : Bool;
      direction : Bool;
      speed : Real;
      angle : Real;
      torque : Real;
      carSpeed : Real;
   END_VAR
   VAR_TEMP   // added for the SCL form of the ladder/FBD networks
      _w1 : Bool;
      _w2 : Bool;
      _w3 : Bool;
      _w4 : Bool;
      _w5 : Bool;
      _w6 : Bool;
      _w7 : Bool;
      _w8 : Bool;
   END_VAR
BEGIN

REGION Network 1: 给上位机下达启动信号
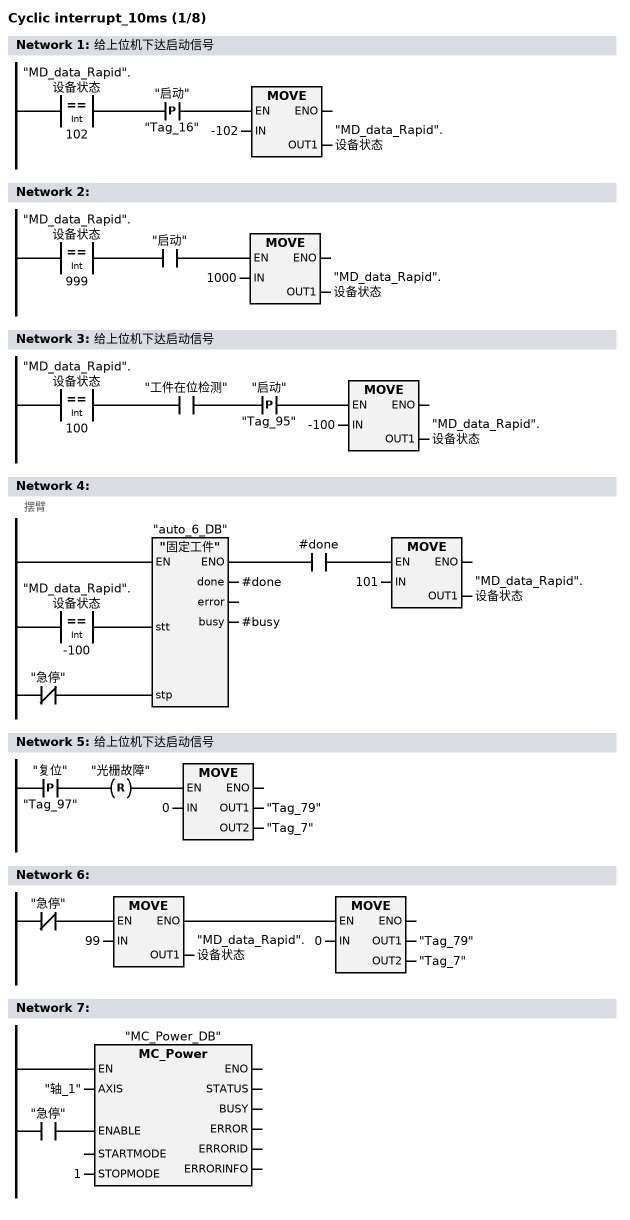
   RUNG wire#powerrail
      { S7_Templates := "SrcType := Int" } EQ_Contact(in1 := "MD_data_Rapid".设备状态, in2 := 102)
      P_Contact(operand := "启动", bit := "Tag_16")
      Move(in := -102, out1 => "MD_data_Rapid".设备状态)
   END_RUNG
   // the same network as SCL:
   #_w1 := ("MD_data_Rapid".设备状态 = 102) AND "启动" AND NOT "Tag_16";   // rising edge of "启动"
   "Tag_16" := "启动";
   IF #_w1 THEN "MD_data_Rapid".设备状态 := -102; END_IF;
END_REGION

REGION Network 2
   RUNG wire#powerrail
      { S7_Templates := "SrcType := Int" } EQ_Contact(in1 := "MD_data_Rapid".设备状态, in2 := 999)
      Contact( "启动" )
      Move(in := 1000, out1 => "MD_data_Rapid".设备状态)
   END_RUNG
   // the same network as SCL:
   IF ("MD_data_Rapid".设备状态 = 999) AND "启动" THEN "MD_data_Rapid".设备状态 := 1000; END_IF;
END_REGION

REGION Network 3: 给上位机下达启动信号
   RUNG wire#powerrail
      { S7_Templates := "SrcType := Int" } EQ_Contact(in1 := "MD_data_Rapid".设备状态, in2 := 100)
      Contact( "工件在位检测" )
      P_Contact(operand := "启动", bit := "Tag_95")
      Move(in := -100, out1 => "MD_data_Rapid".设备状态)
   END_RUNG
   // the same network as SCL:
   #_w1 := ("MD_data_Rapid".设备状态 = 100) AND "工件在位检测" AND "启动" AND NOT "Tag_95";   // rising edge of "启动"
   "Tag_95" := "启动";
   IF #_w1 THEN "MD_data_Rapid".设备状态 := -100; END_IF;
END_REGION

REGION Network 4
   // 摆臂
   RUNG wire#powerrail
      "auto_6_DB"(stt := wire#w1, stp := wire#w2, done => #done, error =>, busy => #busy)
      Contact( #done )
      Move(in := 101, out1 => "MD_data_Rapid".设备状态)
   END_RUNG
   RUNG wire#powerrail
      { S7_Templates := "SrcType := Int" } EQ_Contact(in1 := "MD_data_Rapid".设备状态, in2 := -100)
   END_RUNG wire#w1
   RUNG wire#powerrail
      I_Contact( "急停" )
   END_RUNG wire#w2
   // the same network as SCL:
   "auto_6_DB"(stt := "MD_data_Rapid".设备状态 = (-100), stp := NOT "急停", done => #done, busy => #busy, ENO => #_w1);   // "固定工件"
   IF #_w1 AND #done THEN "MD_data_Rapid".设备状态 := 101; END_IF;
END_REGION

REGION Network 5: 给上位机下达启动信号
   RUNG wire#powerrail
      P_Contact(operand := "复位", bit := "Tag_97")
      R_Coil( "光栅故障" )
      Move(in := 0, out1 => "Tag_79", out2 => "Tag_7")
   END_RUNG
   // the same network as SCL:
   #_w1 := "复位" AND NOT "Tag_97";   // rising edge of "复位"
   "Tag_97" := "复位";
   IF #_w1 THEN
       "光栅故障" := FALSE;
       "Tag_79" := 0;
       "Tag_7" := 0;
   END_IF;
END_REGION

REGION Network 6
   RUNG wire#powerrail
      I_Contact( "急停" )
      Move(in := 99, out1 => "MD_data_Rapid".设备状态)
      Move(in := 0, out1 => "Tag_79", out2 => "Tag_7")
   END_RUNG
   // the same network as SCL:
   IF NOT "急停" THEN
       "MD_data_Rapid".设备状态 := 99;
       "Tag_79" := 0;
       "Tag_7" := 0;
   END_IF;
END_REGION

REGION Network 7
   "MC_Power_DB"(Axis := "轴_1", Enable := "急停", StopMode := 1);   // MC_Power
END_REGION

REGION Network 8
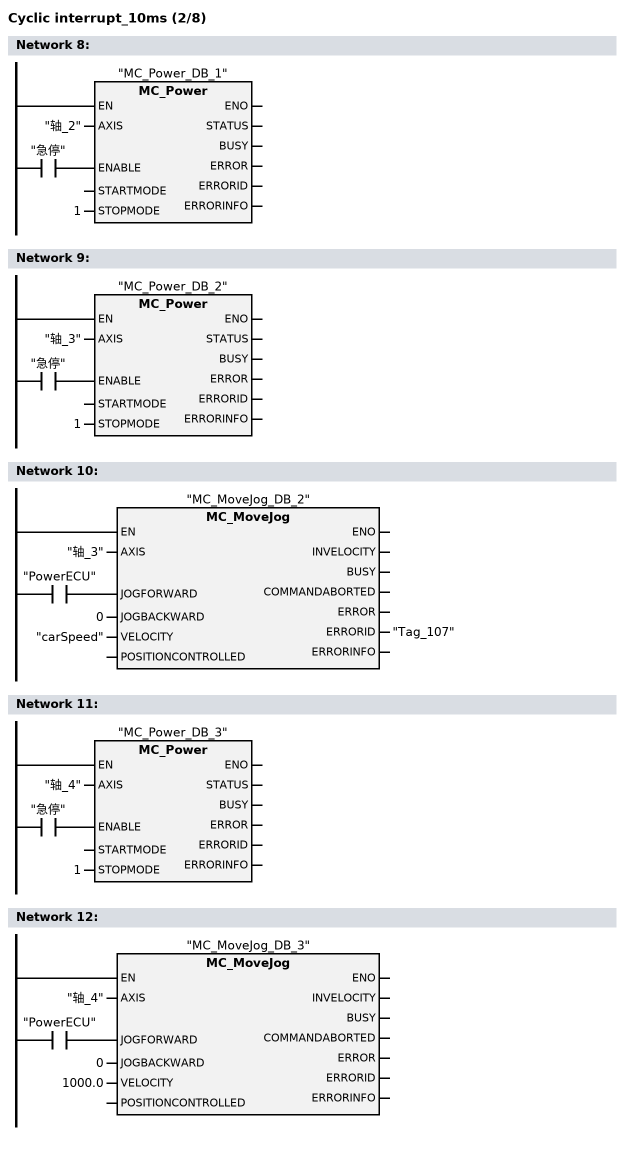
   "MC_Power_DB_1"(Axis := "轴_2", Enable := "急停", StopMode := 1);   // MC_Power
END_REGION

REGION Network 9
   "MC_Power_DB_2"(Axis := "轴_3", Enable := "急停", StopMode := 1);   // MC_Power
END_REGION

REGION Network 10
   "MC_MoveJog_DB_2"(Axis := "轴_3",   // MC_MoveJog
                     JogForward := "PowerECU",
                     JogBackward := 0,
                     Velocity := "carSpeed",
                     ErrorID => "Tag_107");
END_REGION

REGION Network 11
   "MC_Power_DB_3"(Axis := "轴_4", Enable := "急停", StopMode := 1);   // MC_Power
END_REGION

REGION Network 12
   "MC_MoveJog_DB_3"(Axis := "轴_4", JogForward := "PowerECU", JogBackward := 0, Velocity := 1000.0);   // MC_MoveJog
END_REGION

REGION Network 13
   // input move
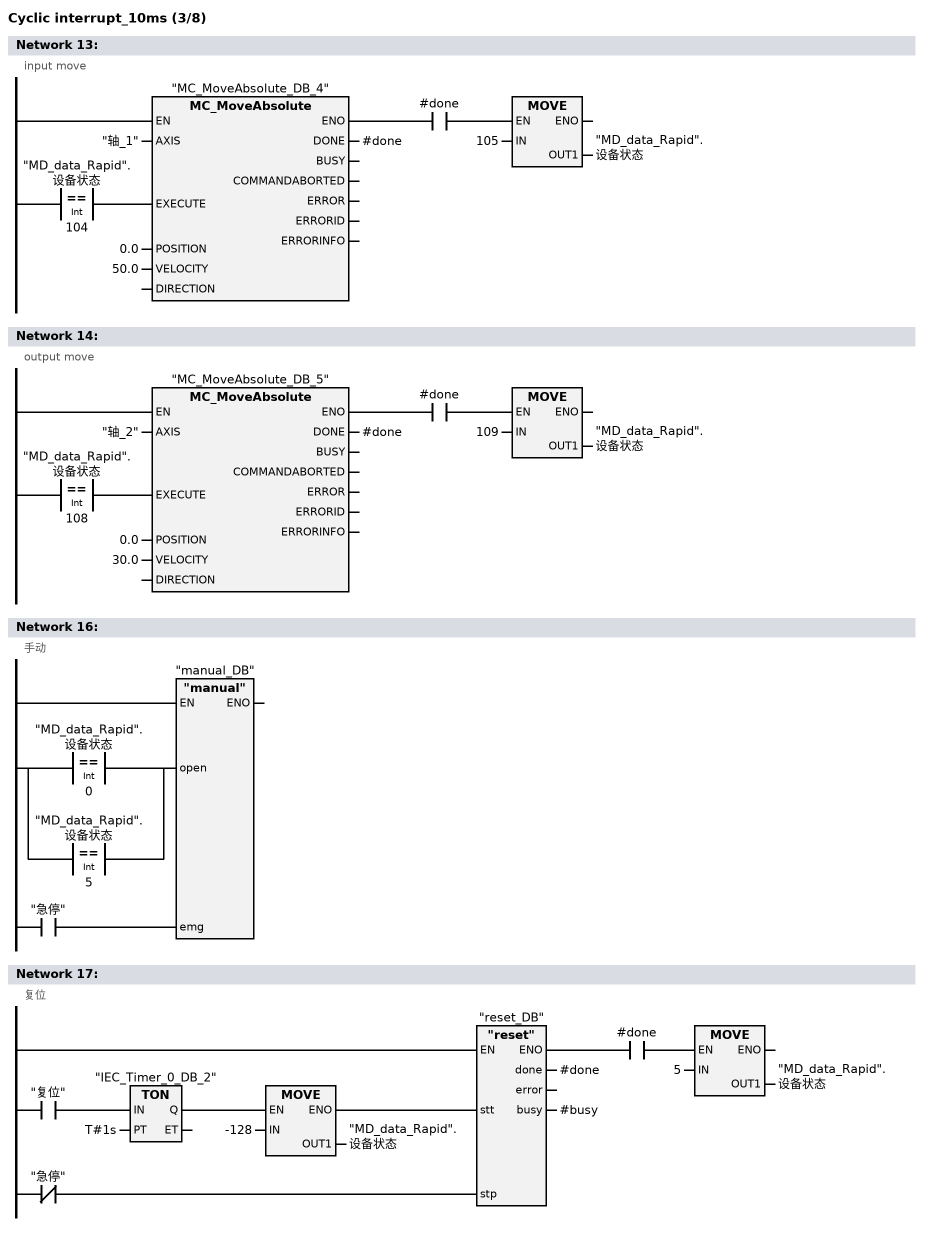
   // ENO of a box is taken as its EN; it also drops when the box reports an error
   "MC_MoveAbsolute_DB_4"(Axis := "轴_1",   // MC_MoveAbsolute
                          Execute := "MD_data_Rapid".设备状态 = 104,
                          Position := 0.0,
                          Velocity := 50.0,
                          Done => #done);
   IF #done THEN "MD_data_Rapid".设备状态 := 105; END_IF;
END_REGION

REGION Network 14
   // output move
   // ENO of a box is taken as its EN; it also drops when the box reports an error
   "MC_MoveAbsolute_DB_5"(Axis := "轴_2",   // MC_MoveAbsolute
                          Execute := "MD_data_Rapid".设备状态 = 108,
                          Position := 0.0,
                          Velocity := 30.0,
                          Done => #done);
   IF #done THEN "MD_data_Rapid".设备状态 := 109; END_IF;
END_REGION

REGION Network 16
   // 手动
   RUNG wire#powerrail
      "manual_DB"(open := wire#w1, emg := wire#w2)
   END_RUNG
   RUNG wire#powerrail
      { S7_Templates := "SrcType := Int" } EQ_Contact(in1 := "MD_data_Rapid".设备状态, in2 := 0)
   END_RUNG wire#w1
   RUNG wire#powerrail
      { S7_Templates := "SrcType := Int" } EQ_Contact(in1 := "MD_data_Rapid".设备状态, in2 := 5)
   END_RUNG wire#w1
   RUNG wire#powerrail
      Contact( "急停" )
   END_RUNG wire#w2
   // the same network as SCL:
   "manual_DB"(open := ("MD_data_Rapid".设备状态 = 0) OR ("MD_data_Rapid".设备状态 = 5), emg := "急停");   // "manual"
END_REGION

REGION Network 17
   // 复位
   "IEC_Timer_0_DB_2".TON(IN := "复位", PT := T#1s);
   IF "IEC_Timer_0_DB_2".Q THEN "MD_data_Rapid".设备状态 := -128; END_IF;
   "reset_DB"(stt := "IEC_Timer_0_DB_2".Q, stp := NOT "急停", done => #done, busy => #busy, ENO => #_w1);   // "reset"
   IF #_w1 AND #done THEN "MD_data_Rapid".设备状态 := 5; END_IF;
END_REGION

REGION Network 18
   // 套上花健
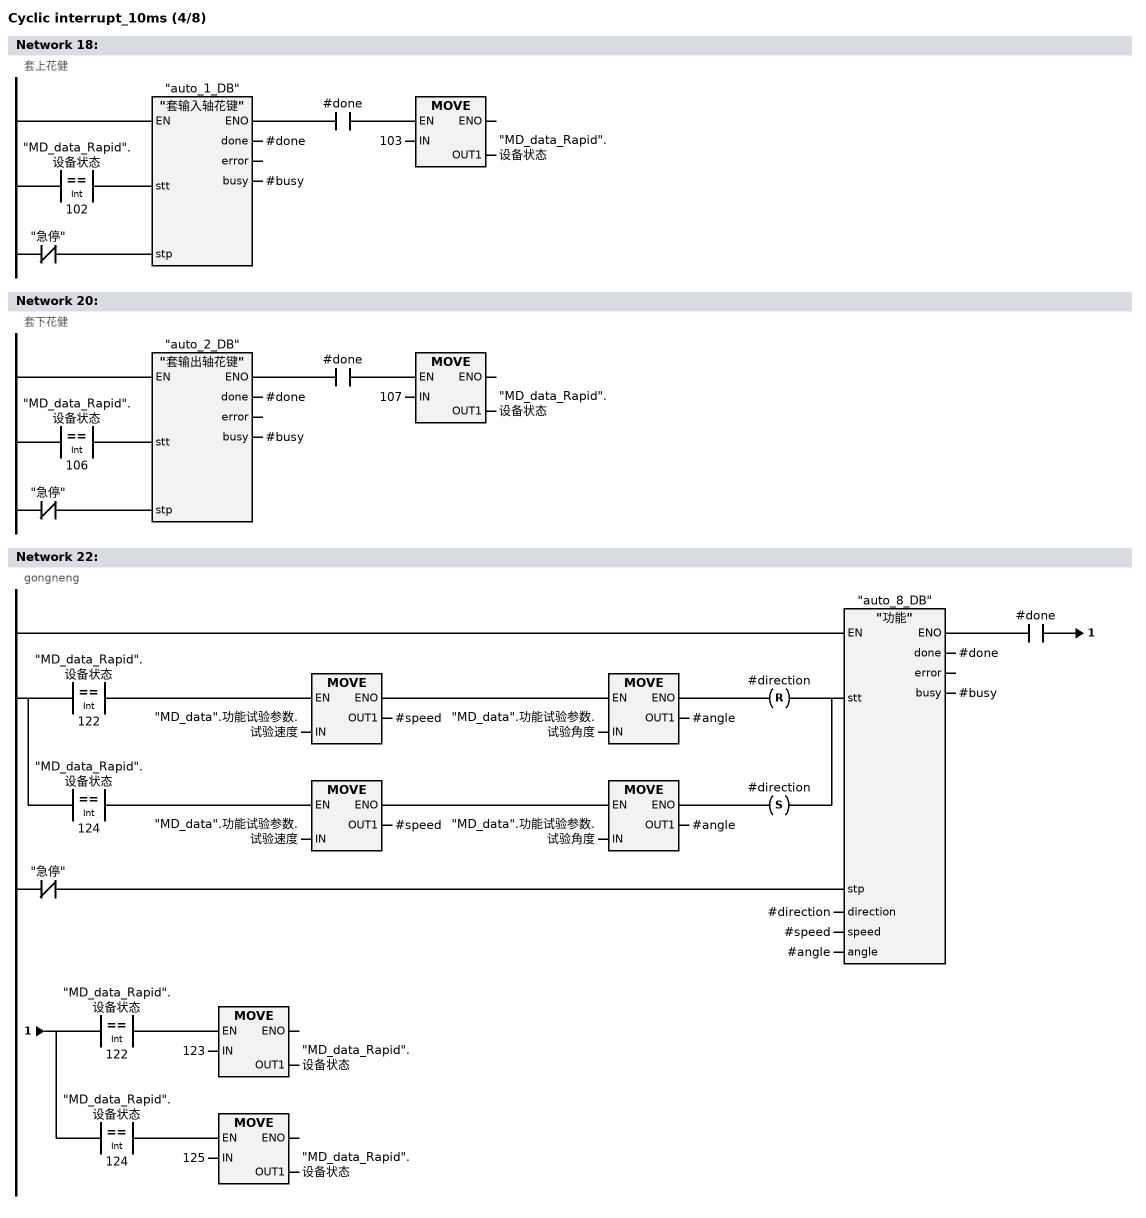
   RUNG wire#powerrail
      "auto_1_DB"(stt := wire#w1, stp := wire#w2, done => #done, error =>, busy => #busy)
      Contact( #done )
      Move(in := 103, out1 => "MD_data_Rapid".设备状态)
   END_RUNG
   RUNG wire#powerrail
      { S7_Templates := "SrcType := Int" } EQ_Contact(in1 := "MD_data_Rapid".设备状态, in2 := 102)
   END_RUNG wire#w1
   RUNG wire#powerrail
      I_Contact( "急停" )
   END_RUNG wire#w2
   // the same network as SCL:
   "auto_1_DB"(stt := "MD_data_Rapid".设备状态 = 102, stp := NOT "急停", done => #done, busy => #busy, ENO => #_w1);   // "套输入轴花键"
   IF #_w1 AND #done THEN "MD_data_Rapid".设备状态 := 103; END_IF;
END_REGION

REGION Network 20
   // 套下花健
   RUNG wire#powerrail
      "auto_2_DB"(stt := wire#w1, stp := wire#w2, done => #done, error =>, busy => #busy)
      Contact( #done )
      Move(in := 107, out1 => "MD_data_Rapid".设备状态)
   END_RUNG
   RUNG wire#powerrail
      { S7_Templates := "SrcType := Int" } EQ_Contact(in1 := "MD_data_Rapid".设备状态, in2 := 106)
   END_RUNG wire#w1
   RUNG wire#powerrail
      I_Contact( "急停" )
   END_RUNG wire#w2
   // the same network as SCL:
   "auto_2_DB"(stt := "MD_data_Rapid".设备状态 = 106, stp := NOT "急停", done => #done, busy => #busy, ENO => #_w1);   // "套输出轴花键"
   IF #_w1 AND #done THEN "MD_data_Rapid".设备状态 := 107; END_IF;
END_REGION

REGION Network 22
   // gongneng
   RUNG wire#powerrail
      "auto_8_DB"(stt := wire#w1, stp := wire#w2, direction := #direction, speed := #speed, angle := #angle, done => #done, error =>, busy => #busy)
      Contact( #done )
      wire#w3
      { S7_Templates := "SrcType := Int" } EQ_Contact(in1 := "MD_data_Rapid".设备状态, in2 := 122)
      Move(in := 123, out1 => "MD_data_Rapid".设备状态)
   END_RUNG
   RUNG wire#powerrail
      { S7_Templates := "SrcType := Int" } EQ_Contact(in1 := "MD_data_Rapid".设备状态, in2 := 122)
      Move(in := "MD_data".功能试验参数.试验速度, out1 => #speed)
      Move(in := "MD_data".功能试验参数.试验角度, out1 => #angle)
      R_Coil( #direction )
   END_RUNG wire#w1
   RUNG wire#powerrail
      { S7_Templates := "SrcType := Int" } EQ_Contact(in1 := "MD_data_Rapid".设备状态, in2 := 124)
      Move(in := "MD_data".功能试验参数.试验速度, out1 => #speed)
      Move(in := "MD_data".功能试验参数.试验角度, out1 => #angle)
      S_Coil( #direction )
   END_RUNG wire#w1
   RUNG wire#powerrail
      I_Contact( "急停" )
   END_RUNG wire#w2
   RUNG wire#w3
      { S7_Templates := "SrcType := Int" } EQ_Contact(in1 := "MD_data_Rapid".设备状态, in2 := 124)
      Move(in := 125, out1 => "MD_data_Rapid".设备状态)
   END_RUNG
   // the same network as SCL:
   #_w1 := "MD_data_Rapid".设备状态 = 122;
   IF #_w1 THEN
       #speed := "MD_data".功能试验参数.试验速度;
       #angle := "MD_data".功能试验参数.试验角度;
       #direction := FALSE;
   END_IF;
   #_w2 := "MD_data_Rapid".设备状态 = 124;
   IF #_w2 THEN
       #speed := "MD_data".功能试验参数.试验速度;
       #angle := "MD_data".功能试验参数.试验角度;
       #direction := TRUE;
   END_IF;
   "auto_8_DB"(stt := #_w1 OR #_w2,   // "功能"
               stp := NOT "急停",
               direction := #direction,
               speed := #speed,
               angle := #angle,
               done => #done,
               busy => #busy,
               ENO => #_w3);
   #_w4 := #_w3 AND #done;
   IF #_w4 AND ("MD_data_Rapid".设备状态 = 122) THEN "MD_data_Rapid".设备状态 := 123; END_IF;
   IF #_w4 AND ("MD_data_Rapid".设备状态 = 124) THEN "MD_data_Rapid".设备状态 := 125; END_IF;
END_REGION

REGION Network 24
   // 空载
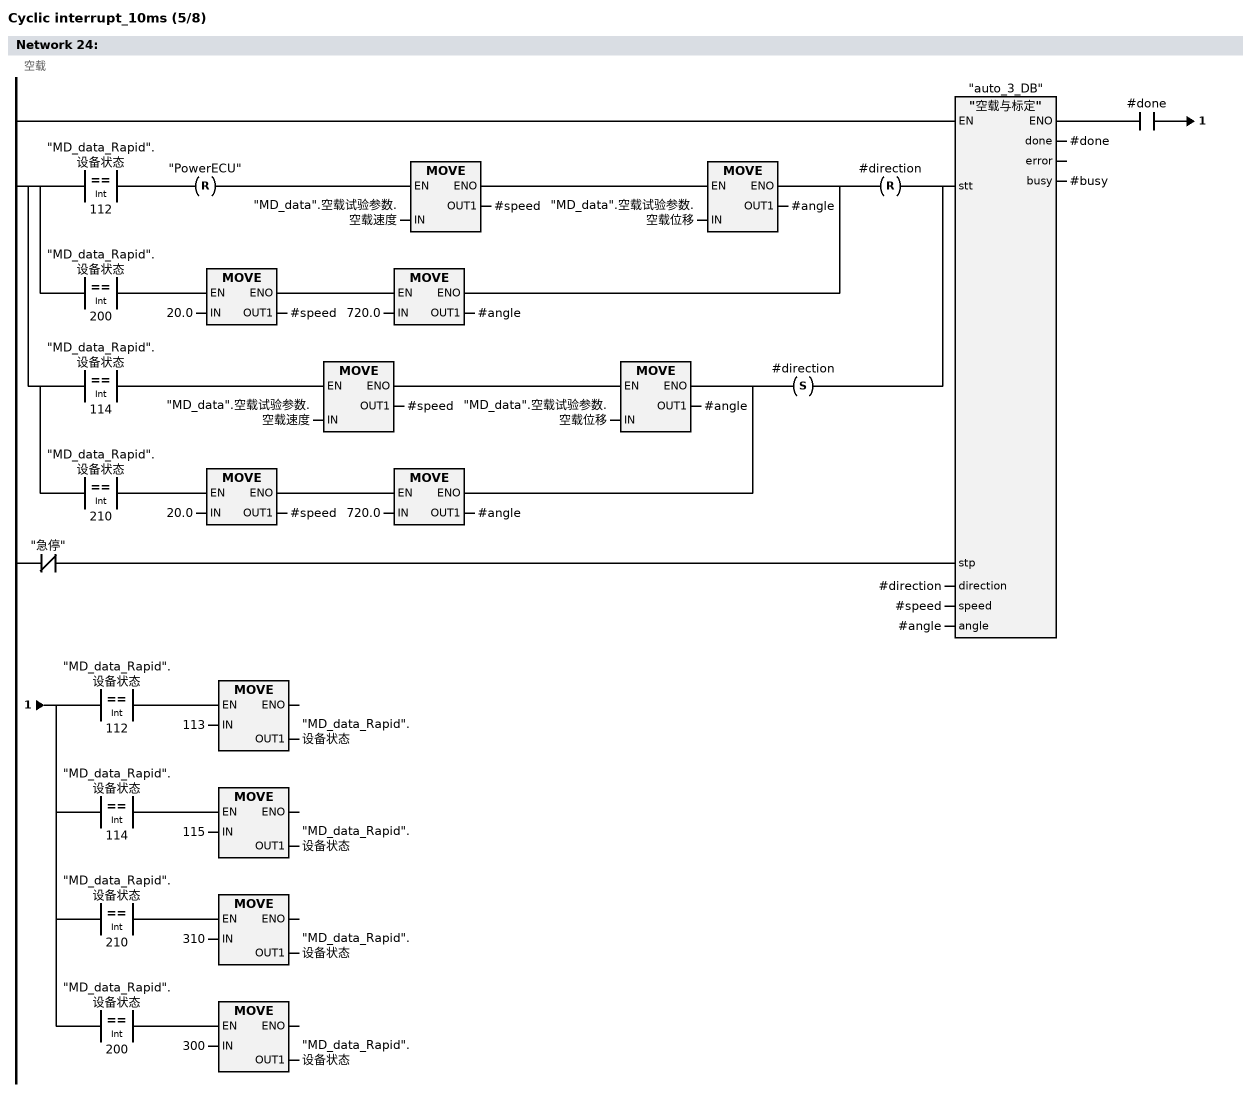
   RUNG wire#powerrail
      "auto_3_DB"(stt := wire#w3, stp := wire#w4, direction := #direction, speed := #speed, angle := #angle, done => #done, error =>, busy => #busy)
      Contact( #done )
      wire#w5
      { S7_Templates := "SrcType := Int" } EQ_Contact(in1 := "MD_data_Rapid".设备状态, in2 := 112)
      Move(in := 113, out1 => "MD_data_Rapid".设备状态)
   END_RUNG
   RUNG wire#powerrail
      { S7_Templates := "SrcType := Int" } EQ_Contact(in1 := "MD_data_Rapid".设备状态, in2 := 112)
      R_Coil( "PowerECU" )
      Move(in := "MD_data".空载试验参数.空载速度, out1 => #speed)
      Move(in := "MD_data".空载试验参数.空载位移, out1 => #angle)
      wire#w1
      R_Coil( #direction )
   END_RUNG wire#w3
   RUNG wire#powerrail
      { S7_Templates := "SrcType := Int" } EQ_Contact(in1 := "MD_data_Rapid".设备状态, in2 := 200)
      Move(in := 20.0, out1 => #speed)
      Move(in := 720.0, out1 => #angle)
   END_RUNG wire#w1
   RUNG wire#powerrail
      { S7_Templates := "SrcType := Int" } EQ_Contact(in1 := "MD_data_Rapid".设备状态, in2 := 114)
      Move(in := "MD_data".空载试验参数.空载速度, out1 => #speed)
      Move(in := "MD_data".空载试验参数.空载位移, out1 => #angle)
      wire#w2
      S_Coil( #direction )
   END_RUNG wire#w3
   RUNG wire#powerrail
      { S7_Templates := "SrcType := Int" } EQ_Contact(in1 := "MD_data_Rapid".设备状态, in2 := 210)
      Move(in := 20.0, out1 => #speed)
      Move(in := 720.0, out1 => #angle)
   END_RUNG wire#w2
   RUNG wire#powerrail
      I_Contact( "急停" )
   END_RUNG wire#w4
   RUNG wire#w5
      { S7_Templates := "SrcType := Int" } EQ_Contact(in1 := "MD_data_Rapid".设备状态, in2 := 114)
      Move(in := 115, out1 => "MD_data_Rapid".设备状态)
   END_RUNG
   RUNG wire#w5
      { S7_Templates := "SrcType := Int" } EQ_Contact(in1 := "MD_data_Rapid".设备状态, in2 := 210)
      Move(in := 310, out1 => "MD_data_Rapid".设备状态)
   END_RUNG
   RUNG wire#w5
      { S7_Templates := "SrcType := Int" } EQ_Contact(in1 := "MD_data_Rapid".设备状态, in2 := 200)
      Move(in := 300, out1 => "MD_data_Rapid".设备状态)
   END_RUNG
   // the same network as SCL:
   #_w1 := "MD_data_Rapid".设备状态 = 112;
   IF #_w1 THEN
       "PowerECU" := FALSE;
       #speed := "MD_data".空载试验参数.空载速度;
       #angle := "MD_data".空载试验参数.空载位移;
   END_IF;
   #_w2 := "MD_data_Rapid".设备状态 = 200;
   IF #_w2 THEN
       #speed := 20.0;
       #angle := 720.0;
   END_IF;
   #_w3 := #_w1 OR #_w2;
   IF #_w3 THEN #direction := FALSE; END_IF;
   #_w4 := "MD_data_Rapid".设备状态 = 114;
   IF #_w4 THEN
       #speed := "MD_data".空载试验参数.空载速度;
       #angle := "MD_data".空载试验参数.空载位移;
   END_IF;
   #_w5 := "MD_data_Rapid".设备状态 = 210;
   IF #_w5 THEN
       #speed := 20.0;
       #angle := 720.0;
   END_IF;
   #_w6 := #_w4 OR #_w5;
   IF #_w6 THEN #direction := TRUE; END_IF;
   "auto_3_DB"(stt := #_w3 OR #_w6,   // "空载与标定"
               stp := NOT "急停",
               direction := #direction,
               speed := #speed,
               angle := #angle,
               done => #done,
               busy => #busy,
               ENO => #_w7);
   #_w8 := #_w7 AND #done;
   IF #_w8 AND ("MD_data_Rapid".设备状态 = 112) THEN "MD_data_Rapid".设备状态 := 113; END_IF;
   IF #_w8 AND ("MD_data_Rapid".设备状态 = 114) THEN "MD_data_Rapid".设备状态 := 115; END_IF;
   IF #_w8 AND ("MD_data_Rapid".设备状态 = 210) THEN "MD_data_Rapid".设备状态 := 310; END_IF;
   IF #_w8 AND ("MD_data_Rapid".设备状态 = 200) THEN "MD_data_Rapid".设备状态 := 300; END_IF;
END_REGION

REGION Network 25
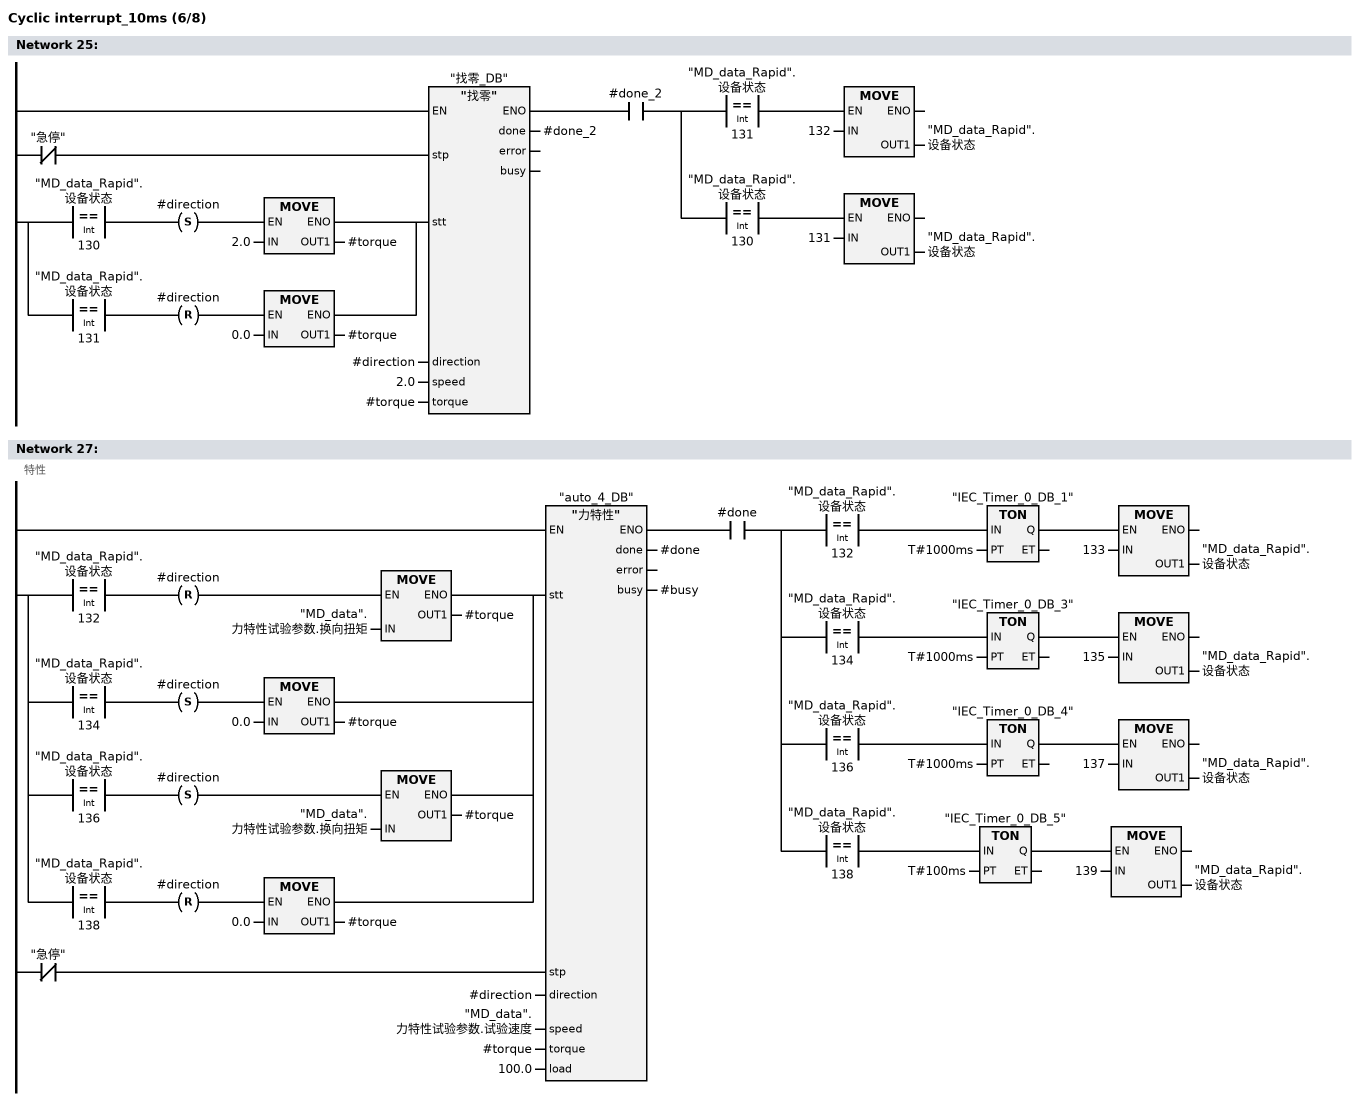
   RUNG wire#powerrail
      "找零_DB"(stp := wire#w1, stt := wire#w2, direction := #direction, speed := 2.0, torque := #torque, done => #done_2, error =>, busy =>)
      Contact( #done_2 )
      wire#w3
      { S7_Templates := "SrcType := Int" } EQ_Contact(in1 := "MD_data_Rapid".设备状态, in2 := 131)
      Move(in := 132, out1 => "MD_data_Rapid".设备状态)
   END_RUNG
   RUNG wire#powerrail
      I_Contact( "急停" )
   END_RUNG wire#w1
   RUNG wire#powerrail
      { S7_Templates := "SrcType := Int" } EQ_Contact(in1 := "MD_data_Rapid".设备状态, in2 := 130)
      S_Coil( #direction )
      Move(in := 2.0, out1 => #torque)
   END_RUNG wire#w2
   RUNG wire#powerrail
      { S7_Templates := "SrcType := Int" } EQ_Contact(in1 := "MD_data_Rapid".设备状态, in2 := 131)
      R_Coil( #direction )
      Move(in := 0.0, out1 => #torque)
   END_RUNG wire#w2
   RUNG wire#w3
      { S7_Templates := "SrcType := Int" } EQ_Contact(in1 := "MD_data_Rapid".设备状态, in2 := 130)
      Move(in := 131, out1 => "MD_data_Rapid".设备状态)
   END_RUNG
   // the same network as SCL:
   #_w1 := "MD_data_Rapid".设备状态 = 130;
   IF #_w1 THEN
       #direction := TRUE;
       #torque := 2.0;
   END_IF;
   #_w2 := "MD_data_Rapid".设备状态 = 131;
   IF #_w2 THEN
       #direction := FALSE;
       #torque := 0.0;
   END_IF;
   "找零_DB"(stp := NOT "急停",   // "找零"
           stt := #_w1 OR #_w2,
           direction := #direction,
           speed := 2.0,
           torque := #torque,
           done => #done_2,
           ENO => #_w3);
   #_w4 := #_w3 AND #done_2;
   IF #_w4 AND ("MD_data_Rapid".设备状态 = 131) THEN "MD_data_Rapid".设备状态 := 132; END_IF;
   IF #_w4 AND ("MD_data_Rapid".设备状态 = 130) THEN "MD_data_Rapid".设备状态 := 131; END_IF;
END_REGION

REGION Network 27
   // 特性
   #_w1 := "MD_data_Rapid".设备状态 = 132;
   IF #_w1 THEN
       #direction := FALSE;
       #torque := "MD_data".力特性试验参数.换向扭矩;
   END_IF;
   #_w2 := "MD_data_Rapid".设备状态 = 134;
   IF #_w2 THEN
       #direction := TRUE;
       #torque := 0.0;
   END_IF;
   #_w3 := "MD_data_Rapid".设备状态 = 136;
   IF #_w3 THEN
       #direction := TRUE;
       #torque := "MD_data".力特性试验参数.换向扭矩;
   END_IF;
   #_w4 := "MD_data_Rapid".设备状态 = 138;
   IF #_w4 THEN
       #direction := FALSE;
       #torque := 0.0;
   END_IF;
   "auto_4_DB"(stt := #_w1 OR #_w2 OR #_w3 OR #_w4,   // "力特性"
               stp := NOT "急停",
               direction := #direction,
               speed := "MD_data".力特性试验参数.试验速度,
               torque := #torque,
               load := 100.0,
               done => #done,
               busy => #busy,
               ENO => #_w5);
   #_w6 := #_w5 AND #done;
   "IEC_Timer_0_DB_1".TON(IN := #_w6 AND ("MD_data_Rapid".设备状态 = 132), PT := T#1000ms);
   IF "IEC_Timer_0_DB_1".Q THEN "MD_data_Rapid".设备状态 := 133; END_IF;
   "IEC_Timer_0_DB_3".TON(IN := #_w6 AND ("MD_data_Rapid".设备状态 = 134), PT := T#1000ms);
   IF "IEC_Timer_0_DB_3".Q THEN "MD_data_Rapid".设备状态 := 135; END_IF;
   "IEC_Timer_0_DB_4".TON(IN := #_w6 AND ("MD_data_Rapid".设备状态 = 136), PT := T#1000ms);
   IF "IEC_Timer_0_DB_4".Q THEN "MD_data_Rapid".设备状态 := 137; END_IF;
   "IEC_Timer_0_DB_5".TON(IN := #_w6 AND ("MD_data_Rapid".设备状态 = 138), PT := T#100ms);
   IF "IEC_Timer_0_DB_5".Q THEN "MD_data_Rapid".设备状态 := 139; END_IF;
END_REGION

REGION Network 29
   // 逆向空载
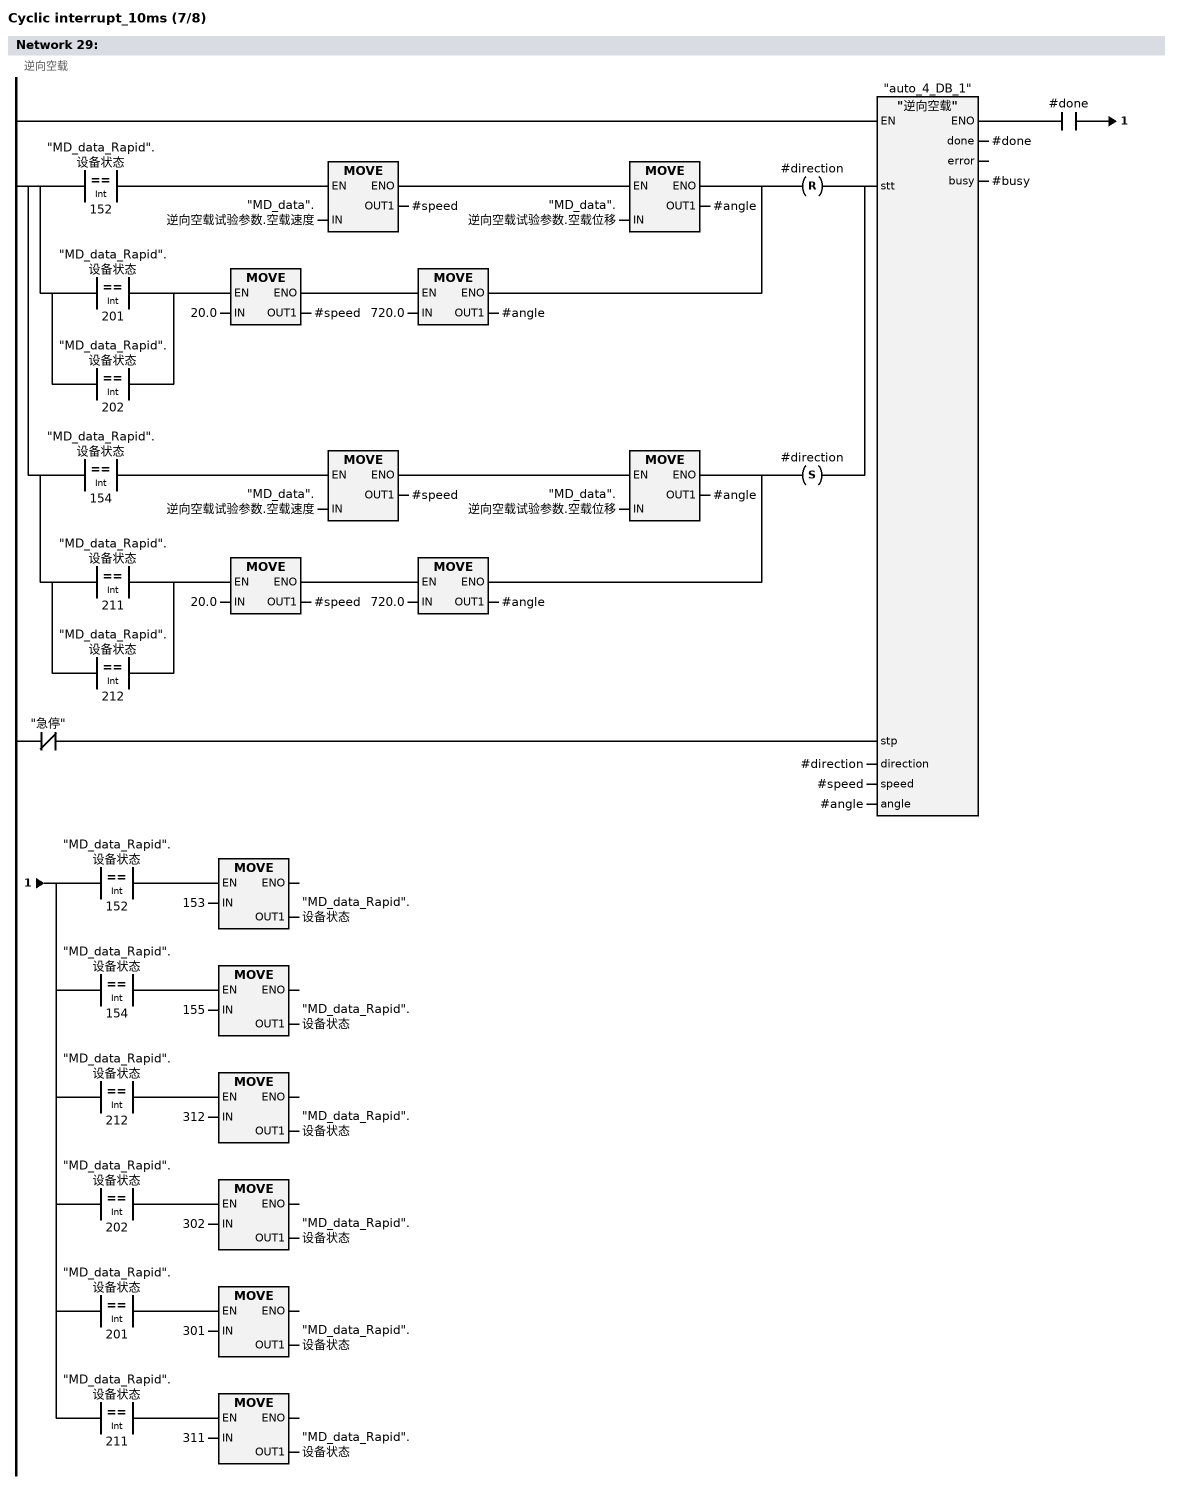
   RUNG wire#powerrail
      "auto_4_DB_1"(stt := wire#w5, stp := wire#w6, direction := #direction, speed := #speed, angle := #angle, done => #done, error =>, busy => #busy)
      Contact( #done )
      wire#w7
      { S7_Templates := "SrcType := Int" } EQ_Contact(in1 := "MD_data_Rapid".设备状态, in2 := 152)
      Move(in := 153, out1 => "MD_data_Rapid".设备状态)
   END_RUNG
   RUNG wire#powerrail
      { S7_Templates := "SrcType := Int" } EQ_Contact(in1 := "MD_data_Rapid".设备状态, in2 := 152)
      Move(in := "MD_data".逆向空载试验参数.空载速度, out1 => #speed)
      Move(in := "MD_data".逆向空载试验参数.空载位移, out1 => #angle)
      wire#w1
      R_Coil( #direction )
   END_RUNG wire#w5
   RUNG wire#powerrail
      { S7_Templates := "SrcType := Int" } EQ_Contact(in1 := "MD_data_Rapid".设备状态, in2 := 201)
      wire#w2
      Move(in := 20.0, out1 => #speed)
      Move(in := 720.0, out1 => #angle)
   END_RUNG wire#w1
   RUNG wire#powerrail
      { S7_Templates := "SrcType := Int" } EQ_Contact(in1 := "MD_data_Rapid".设备状态, in2 := 202)
   END_RUNG wire#w2
   RUNG wire#powerrail
      { S7_Templates := "SrcType := Int" } EQ_Contact(in1 := "MD_data_Rapid".设备状态, in2 := 154)
      Move(in := "MD_data".逆向空载试验参数.空载速度, out1 => #speed)
      Move(in := "MD_data".逆向空载试验参数.空载位移, out1 => #angle)
      wire#w3
      S_Coil( #direction )
   END_RUNG wire#w5
   RUNG wire#powerrail
      { S7_Templates := "SrcType := Int" } EQ_Contact(in1 := "MD_data_Rapid".设备状态, in2 := 211)
      wire#w4
      Move(in := 20.0, out1 => #speed)
      Move(in := 720.0, out1 => #angle)
   END_RUNG wire#w3
   RUNG wire#powerrail
      { S7_Templates := "SrcType := Int" } EQ_Contact(in1 := "MD_data_Rapid".设备状态, in2 := 212)
   END_RUNG wire#w4
   RUNG wire#powerrail
      I_Contact( "急停" )
   END_RUNG wire#w6
   RUNG wire#w7
      { S7_Templates := "SrcType := Int" } EQ_Contact(in1 := "MD_data_Rapid".设备状态, in2 := 154)
      Move(in := 155, out1 => "MD_data_Rapid".设备状态)
   END_RUNG
   RUNG wire#w7
      { S7_Templates := "SrcType := Int" } EQ_Contact(in1 := "MD_data_Rapid".设备状态, in2 := 212)
      Move(in := 312, out1 => "MD_data_Rapid".设备状态)
   END_RUNG
   RUNG wire#w7
      { S7_Templates := "SrcType := Int" } EQ_Contact(in1 := "MD_data_Rapid".设备状态, in2 := 202)
      Move(in := 302, out1 => "MD_data_Rapid".设备状态)
   END_RUNG
   RUNG wire#w7
      { S7_Templates := "SrcType := Int" } EQ_Contact(in1 := "MD_data_Rapid".设备状态, in2 := 201)
      Move(in := 301, out1 => "MD_data_Rapid".设备状态)
   END_RUNG
   RUNG wire#w7
      { S7_Templates := "SrcType := Int" } EQ_Contact(in1 := "MD_data_Rapid".设备状态, in2 := 211)
      Move(in := 311, out1 => "MD_data_Rapid".设备状态)
   END_RUNG
   // the same network as SCL:
   #_w1 := "MD_data_Rapid".设备状态 = 152;
   IF #_w1 THEN
       #speed := "MD_data".逆向空载试验参数.空载速度;
       #angle := "MD_data".逆向空载试验参数.空载位移;
   END_IF;
   #_w2 := ("MD_data_Rapid".设备状态 = 201) OR ("MD_data_Rapid".设备状态 = 202);
   IF #_w2 THEN
       #speed := 20.0;
       #angle := 720.0;
   END_IF;
   #_w3 := #_w1 OR #_w2;
   IF #_w3 THEN #direction := FALSE; END_IF;
   #_w4 := "MD_data_Rapid".设备状态 = 154;
   IF #_w4 THEN
       #speed := "MD_data".逆向空载试验参数.空载速度;
       #angle := "MD_data".逆向空载试验参数.空载位移;
   END_IF;
   #_w5 := ("MD_data_Rapid".设备状态 = 211) OR ("MD_data_Rapid".设备状态 = 212);
   IF #_w5 THEN
       #speed := 20.0;
       #angle := 720.0;
   END_IF;
   #_w6 := #_w4 OR #_w5;
   IF #_w6 THEN #direction := TRUE; END_IF;
   "auto_4_DB_1"(stt := #_w3 OR #_w6,   // "逆向空载"
                 stp := NOT "急停",
                 direction := #direction,
                 speed := #speed,
                 angle := #angle,
                 done => #done,
                 busy => #busy,
                 ENO => #_w7);
   #_w8 := #_w7 AND #done;
   IF #_w8 AND ("MD_data_Rapid".设备状态 = 152) THEN "MD_data_Rapid".设备状态 := 153; END_IF;
   IF #_w8 AND ("MD_data_Rapid".设备状态 = 154) THEN "MD_data_Rapid".设备状态 := 155; END_IF;
   IF #_w8 AND ("MD_data_Rapid".设备状态 = 212) THEN "MD_data_Rapid".设备状态 := 312; END_IF;
   IF #_w8 AND ("MD_data_Rapid".设备状态 = 202) THEN "MD_data_Rapid".设备状态 := 302; END_IF;
   IF #_w8 AND ("MD_data_Rapid".设备状态 = 201) THEN "MD_data_Rapid".设备状态 := 301; END_IF;
   IF #_w8 AND ("MD_data_Rapid".设备状态 = 211) THEN "MD_data_Rapid".设备状态 := 311; END_IF;
END_REGION

REGION Network 30
   // 振动
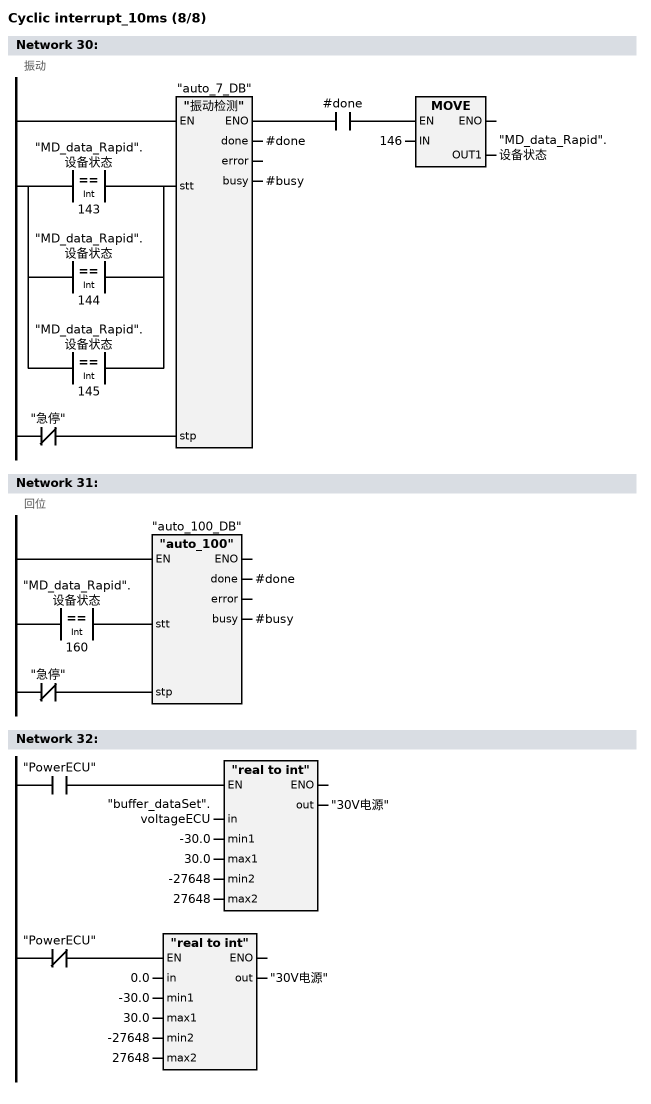
   RUNG wire#powerrail
      "auto_7_DB"(stt := wire#w1, stp := wire#w2, done => #done, error =>, busy => #busy)
      Contact( #done )
      Move(in := 146, out1 => "MD_data_Rapid".设备状态)
   END_RUNG
   RUNG wire#powerrail
      { S7_Templates := "SrcType := Int" } EQ_Contact(in1 := "MD_data_Rapid".设备状态, in2 := 143)
   END_RUNG wire#w1
   RUNG wire#powerrail
      { S7_Templates := "SrcType := Int" } EQ_Contact(in1 := "MD_data_Rapid".设备状态, in2 := 144)
   END_RUNG wire#w1
   RUNG wire#powerrail
      { S7_Templates := "SrcType := Int" } EQ_Contact(in1 := "MD_data_Rapid".设备状态, in2 := 145)
   END_RUNG wire#w1
   RUNG wire#powerrail
      I_Contact( "急停" )
   END_RUNG wire#w2
   // the same network as SCL:
   "auto_7_DB"(stt := ("MD_data_Rapid".设备状态 = 143) OR ("MD_data_Rapid".设备状态 = 144) OR ("MD_data_Rapid".设备状态 = 145),   // "振动检测"
               stp := NOT "急停",
               done => #done,
               busy => #busy,
               ENO => #_w1);
   IF #_w1 AND #done THEN "MD_data_Rapid".设备状态 := 146; END_IF;
END_REGION

REGION Network 31
   // 回位
   RUNG wire#powerrail
      "auto_100_DB"(stt := wire#w1, stp := wire#w2, done => #done, error =>, busy => #busy)
   END_RUNG
   RUNG wire#powerrail
      { S7_Templates := "SrcType := Int" } EQ_Contact(in1 := "MD_data_Rapid".设备状态, in2 := 160)
   END_RUNG wire#w1
   RUNG wire#powerrail
      I_Contact( "急停" )
   END_RUNG wire#w2
   // the same network as SCL:
   "auto_100_DB"(stt := "MD_data_Rapid".设备状态 = 160, stp := NOT "急停", done => #done, busy => #busy);   // "auto_100"
END_REGION

REGION Network 32
   RUNG wire#powerrail
      Contact( "PowerECU" )
      "real to int"(in := "buffer_dataSet".voltageECU, min1 := -30.0, max1 := 30.0, min2 := -27648, max2 := 27648, out => "30V电源")
   END_RUNG
   RUNG wire#powerrail
      I_Contact( "PowerECU" )
      "real to int"(in := 0.0, min1 := -30.0, max1 := 30.0, min2 := -27648, max2 := 27648, out => "30V电源")
   END_RUNG
   // the same network as SCL:
   IF "PowerECU" THEN
       "real to int"(in := "buffer_dataSet".voltageECU,
                     min1 := -30.0,
                     max1 := 30.0,
                     min2 := -27648,
                     max2 := 27648,
                     out => "30V电源");
   END_IF;
   IF NOT "PowerECU" THEN
       "real to int"(in := 0.0, min1 := -30.0, max1 := 30.0, min2 := -27648, max2 := 27648, out => "30V电源");
   END_IF;
END_REGION
END_ORGANIZATION_BLOCK

ORGANIZATION_BLOCK "Cyclic interrupt_500ms"   // OB31, LAD, CyclicInterrupt
{ S7_Optimized_Access := 'TRUE' }
VERSION : 0.1
   VAR_INPUT
      Initial_Call : Bool;   // Initial call of this OB
      Event_Count : Int;   // Events discarded
   END_VAR
BEGIN

REGION Network 1
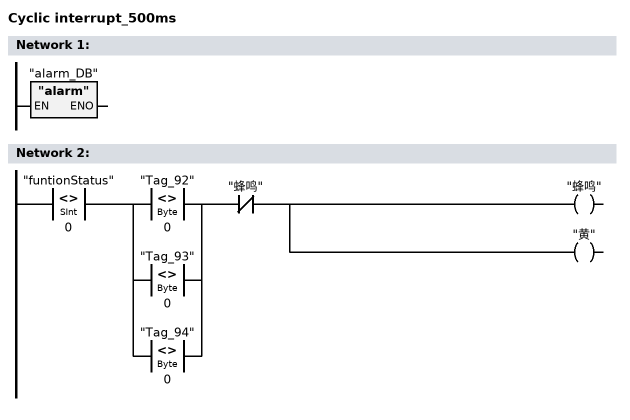
   RUNG wire#powerrail
      "alarm_DB"()
   END_RUNG
   // the same network as SCL:
   "alarm_DB"();   // "alarm"
END_REGION

REGION Network 2
   RUNG wire#powerrail
      { S7_Templates := "SrcType := SInt" } NE_Contact(in1 := "funtionStatus", in2 := 0)
      wire#w1
      { S7_Templates := "SrcType := Byte" } NE_Contact(in1 := "Tag_92", in2 := 0)
      wire#w2
      I_Contact( "蜂鸣" )
      wire#w3
      Coil( "蜂鸣" )
   END_RUNG
   RUNG wire#w1
      { S7_Templates := "SrcType := Byte" } NE_Contact(in1 := "Tag_93", in2 := 0)
   END_RUNG wire#w2
   RUNG wire#w1
      { S7_Templates := "SrcType := Byte" } NE_Contact(in1 := "Tag_94", in2 := 0)
   END_RUNG wire#w2
   RUNG wire#w3
      Coil( "黄" )
   END_RUNG
   // the same network as SCL:
   "蜂鸣" := ("funtionStatus" <> 0) AND (("Tag_92" <> 0) OR ("Tag_93" <> 0) OR ("Tag_94" <> 0)) AND NOT "蜂鸣";
   "黄" := "蜂鸣";
END_REGION
END_ORGANIZATION_BLOCK

ORGANIZATION_BLOCK "Startup"   // OB100, LAD, Startup
TITLE = "Complete Restart"
{ S7_Optimized_Access := 'TRUE' }
VERSION : 0.1
   VAR_INPUT
      LostRetentive : Bool;   // True if retentive data are lost
      LostRTC : Bool;   // True if date and time are lost
   END_VAR
BEGIN

REGION Network 1
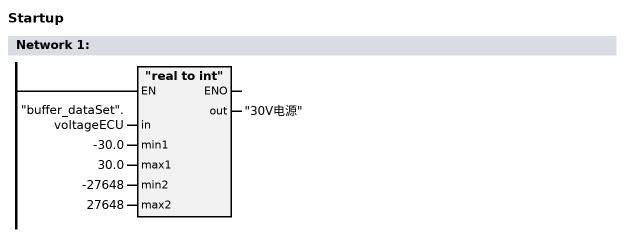
   RUNG wire#powerrail
      "real to int"(in := "buffer_dataSet".voltageECU, min1 := -30.0, max1 := 30.0, min2 := -27648, max2 := 27648, out => "30V电源")
   END_RUNG
   // the same network as SCL:
   "real to int"(in := "buffer_dataSet".voltageECU,
                 min1 := -30.0,
                 max1 := 30.0,
                 min2 := -27648,
                 max2 := 27648,
                 out => "30V电源");
END_REGION
END_ORGANIZATION_BLOCK